(* CODESYS project Dynamixel_V3.2.2.library
   Author: Clément Jaquiéry
   Placeholder: Dynamixel
   Title: Dynamixel
   Version: 3.2.2
   Description: Permet le contrôle de Dynamixels
   Company: CPNV

Project tree, tasks and I/O mapping:
  libraries: Tc2_SerialCom, * (Beckhoff Automation GmbH); Tc2_Standard, * (Beckhoff Automation GmbH); Tc2_System, * (Beckhoff Automation GmbH); Tc2_Utilities, * (Beckhoff Automation GmbH); Tc3_Module, * (Beckhoff Automation GmbH)
  DUTs/
    data type DXL_Error
    data type E_DXL
    data type E_Packet_Status
    data type ST_DXL_Position
    data type ST_SendPacket
  GVLs/
    global variables DXL_Const
  POUs/
    function block FB_CSVRead [ST]
    function block FB_CSVWrite [ST]
    function block FB_DXL [ST]: SetActTorque, SetError, CreatePosition, DeletePosition, DisableTorque, GetActPosition, GetDatabase, Homing, MoveAbs, MovePosition, MoveRel, ReadCSV, RenamePosition, Reset, SetPosition, SetPositionD_Gain, SetPositionI_Gain, SetPositionP_Gain, SetVelocityI_Gain, SetVelocityP_Gain, ToggleTorque, WriteCSV
    function block FB_SyncDXL [ST]: AddDynamixel, ClearDynamixel, MoveAbs, MoveDiffAbs, Reset
    function block FB_U2D2_V3 [ST]: BulkWrite, BulkWriteAdd, HiByte, HiWord, LoByte, LoWord, MakeDWord, MakeWord, SendPacket, SendPacketParam, SendSyncPacket, UpdateCRC, SyncRead, SyncReadAdd, SyncWrite, SyncWriteAdd, Execute, Read, Reboot, RegWrite, SyncReset, Write
*)

// DUTs/DXL_Error
{attribute 'qualified_only'}
{attribute 'strict'}
{attribute 'to_string'}
TYPE DXL_Error :
(
	NoError := 0,
	ExceedCounter,
	ExceedTorque,
	WriteError,
	CSV_Read_Error,
	CSV_Write_Error

)BYTE;
END_TYPE

// DUTs/E_DXL
{attribute 'qualified_only'}
{attribute 'strict'}

// https://emanual.robotis.com/docs/en/dxl/x/

TYPE E_DXL :
(
	Model_Number 			:= 0, //Length 2
	Model_Information		:= 2, //Lenght 4
	Firmware_Version 		:= 6, //Length 4
	ID 						:= 7, //Length 1
	Baud_Rate 				:= 8, //Length 1
	Return_Delay_Time 		:= 9, //Length 1
	Drive_Mode 				:= 10, //Length 1
	Operating_Mode 			:= 11, //Length 1
	Secondary_ID 			:= 12, //Length 1
	Protocol_Type 			:= 13, //Length 1
	Homing_Offset 			:= 20, //Length 4
	Moving_Treshold 		:= 24, //Length 4
	Temperature_Limit 		:= 31, //Length 1
	Max_Voltage_Limit		:= 32, //Length 2
	Min_Voltage_Limit		:= 34, //Length 2
	PWM_Limit				:= 36, //Length 2
	Velocity_Limit			:= 44, //Length 4
	Max_Position_Limit		:= 48, //Length 4
	Min_Position_Limit		:= 52, //Length 4
	Startup_Configuration	:= 60, //Length 1
	Shutdown				:= 63, //Length 1
	Torque_Enable 			:= 64, //Length 1
	LED 					:= 65, //Length 1
	Status_Return_Level 	:= 68, //Length 1
	Registered_Instruction 	:= 69, //Length 1
	Hardware_Error_Status 	:= 70, //Length 1
	Velocity_I_Gain			:= 76, //Length 2
	Velocity_P_Gain			:= 78, //Length 2
	Position_D_Gain			:= 80, //Length 2
	Position_I_Gain			:= 82, //Length 2
	Position_P_Gain			:= 84, //Length 2
	Feedforward_2nd_Gain	:= 88, //Length 2
	Feedforward_1st_Gain	:= 90, //Length 2
	Bus_Watchdog			:= 98, //Length 1
	Goal_PWM				:= 100, //Length 2
	Goal_Velocity			:= 104, //Length 4
	Profile_Acceleration	:= 108, //Length 4
	Profile_Velocity		:= 112, //Length 4
	Goal_Position			:= 116, //Length 4
	Realtime_Tick			:= 120, //Length 2
	Moving					:= 122, //Length 1
	Moving_Status			:= 123, //Length 1
	Present_PWM				:= 124, //Length 2
	Present_Load			:= 126, //Length 2
	Present_Velocity		:= 128, //Length 4
	Present_Position		:= 132, //Length 4
	Velocity_Trajectory		:= 136, //Length 4
	Position_Trajectory		:= 140, //Length 4
	Present_Input_Voltage	:= 144, //Length 2
	Present_Temperature		:= 146, //Length 1
	Backup_Ready			:= 147  //Length 1
)BYTE;
END_TYPE

// DUTs/E_Packet_Status
{attribute 'qualified_only'}
{attribute 'strict'}
TYPE E_Packet_Status : 						// https://emanual.robotis.com/docs/en/dxl/protocol2/
(
	Waiting						:= 0,	
	Send_Result_Fail			:= 1,	// Failed to process the sent Instruction Packet
	Send_Instruction_Error		:= 2,	// An undefined Instruction has been used. Action has been used without Reg Write
	Send_CRC_Error				:= 3,   // The CRC of the sent Packet does not match the expected value
	Send_Data_Range_Error		:= 4,	// Data to be written to the specified Address is outside the range of the minimum/maximum value
	Send_Data_Lenght_Error		:= 5,	// Attempted to write Data that is shorter than the required data length of the specified Address (ex: when you attempt to only use 2 bytes of a register that has been defined as 4 bytes)
	Send_Data_Limit_Error		:= 6,	// Data to be written to the specified Address is outside of the configured Limit value
	Send_Access_Error			:= 7,	// Attempted to write a value to an Address that is Read Only or has not been defined. Attempted to read a value from an Address that is Write Only or has not been defined. Attempted to write a value to an EEPROM register while Torque was Enabled.
	Receive_TimeOut,
	Receive_Instruction_Error,
	Receive_CRC_Error,
	SendByte_Fail,
	Success
)BYTE;
END_TYPE

// DUTs/ST_DXL_Position
TYPE ST_DXL_Position :
STRUCT
	byIndex : BYTE;
	sName	: T_MaxString;
	diPos	: DINT;
END_STRUCT
END_TYPE

// DUTs/ST_SendPacket
TYPE ST_SendPacket :
STRUCT
	eStatus : ARRAY[0..252] OF E_Packet_Status;
	diValue : ARRAY[0..252] OF DINT;
	arPacket : ARRAY[0..MAX_PACKET_LENGTH] OF BYTE;
	wLength : WORD;
	byNumPacketsReceive : BYTE;
END_STRUCT
END_TYPE

// GVLs/DXL_Const
VAR_GLOBAL CONSTANT
	//--------------Paramètres de réglage des dynamixels--------------
	MAX_ERROR : BYTE := 5;						// Nombre d'essais de communication avant de se mettre en erreur
	TIME_TORQUE_ERROR : TIME := T#250MS;		// Temps avant que le dynamixel soit en erreur dû aux couples
	TIME_OUT_PACKET : TIME := T#100MS;			// Temps avant que le dynamixel soit en erreur dû aux non retour de paquet
	//--------------Paramètres de longueurs max de paquets--------------
	MAX_LENGTH_BUFFER : WORD := 74;				// Longueur max de la mémoire tampon d'envois de paquets
	MAX_PACKET_LENGTH : BYTE := 99;				// Longueur max des paquets envoyés
	MAX_RECEIVE_PACKET_LENGTH : WORD := 300;	// Longueur max des paquets reçus
	//--------------Paramètres de longueurs max du tableau--------------
	MAX_CSV_ROWS 			: UDINT := 29;	// |, Longueur du tableau à ajuster pour avoir plus de position
	MAX_CSV_COLUMNS 		: UDINT := 2;	// -, Ne pas toucher
	MAX_CSV_FIELD_LENGTH	: UDINT := 20;	// Ne pas toucher
END_VAR

// POUs/FB_CSVRead
FUNCTION_BLOCK FB_CSVRead(* Reading of CSV file in binary mode. Field values may contain non-printing control characters (binary data or special characters like line feed, carriage return or quotation mark...). *)
VAR	
	nRow	 	: UDINT 	:= 0;(* Row number (record) *)
	nColumn		: UDINT 	:= 0;(* Column number (record field) *)
	cbDone		: UDINT 	:= 0;(* Counts allready parsed data bytes *)
	hFile		: UINT		:= 0;(* File handle of the source file *)
	step		: DWORD 	:= 0;
	fbFileOpen	: FB_FileOpen;(* Opens file *)
	fbFileClose	: FB_FileClose;(* Closes file *)
	fbFileRead	: FB_FileRead;(* Writes binary data *)
	fbReader	: FB_CSVMemBufferReader;(* Helper function block used to parse CSV data bytes *)

	record		: ARRAY[0..1024] OF BYTE;(* Binary row data buffer. The size of this buffer have to be > length of longest record line + 2 (CRLF)  *)
	cbRecord	: UDINT := 0;(* Number of bytes in row buffer *)
	cbField		: UDINT;(* Number of bytes in field buffer *)
END_VAR
VAR_INPUT
	bRead		: BOOL := FALSE;(* Rising edge starts program execution *)
	sNetId		: T_AmsNetId := '';	(* TwinCAT system network address *)
	sFileName	: T_MaxString := '';(* CSV source file path and name *)
	database	: POINTER TO ARRAY[0..MAX_CSV_ROWS] OF ST_DXL_Position;(* Target PLC database *)
END_VAR
VAR_OUTPUT
	bBusy		: BOOL;
	bError		: BOOL;
	nErrId		: UDINT;
END_VAR

CASE step OF
	0:	(* Wait for rising edge at bRead variable *)
		IF bRead THEN
			bRead 	:= FALSE;
			bBusy 	:= TRUE;
			bError	:= FALSE;
			nErrId	:= 0;
			hFile	:= 0;
			nRow	:= 0;
			nColumn	:= 0;
			cbRecord:= 0;
			cbDone 	:= 0;
			step 	:= 1;
		END_IF

	1:	(* Open source file *)
		fbFileOpen(  bExecute := FALSE  );
		fbFileOpen( sNetId := sNetId, sPathName := sFileName, nMode := FOPEN_MODEREAD OR FOPEN_MODEBINARY,(* Open file in BINARY mode! *)
					ePath := PATH_GENERIC, bExecute := TRUE );
		step := 2;

	2:(* Wait until open not busy *)
		fbFileOpen( bExecute := FALSE, bError => bError, nErrID => nErrID, hFile => hFile );
		IF NOT fbFileOpen.bBusy THEN
			IF NOT fbFileOpen.bError THEN
				step := 3;
			ELSE(* Error: file not found? *)
				step := 100;
			END_IF
		END_IF

	3:	(* Read data bytes from file *)
		fbFileRead( bExecute := FALSE );
		fbFileRead( sNetId := sNetId, hFile := hFile, pReadBuff := ADR( record[ cbRecord ] ), cbReadLen := SIZEOF( record ) - cbRecord, bExecute :=TRUE );
		step := 4;

	4:(* Wait until read not busy *)
		fbFileRead( bExecute := FALSE, bError => bError, nErrID => nErrID );
		IF NOT fbFileRead.bBusy THEN
			IF NOT fbFileRead.bError THEN
				IF fbFileRead.bEOF THEN
					step := 10;(* End of file reached => Close source file *)
				ELSE
					cbRecord := cbRecord + fbFileRead.cbRead;(* Recalculate the new size of data buffer *)
					step := 5;(* Parse binary data *)
				END_IF
			ELSE(* Error *)
				step := 100;
			END_IF
		END_IF

	5:(* Parse binary data *)
		cbDone := 0;(* Reset number of parsed data bytes *)
		fbReader.eCmd := eEnumCmd_First;(* Read first field value *)
		REPEAT
			fbReader( pBuffer := ADR( record ), cbBuffer := cbRecord );
			IF fbReader.bOk THEN
				fbReader.eCmd := eEnumCmd_Next;(* Read next field value *)
				cbDone := cbDone + fbReader.cbRead;(* Count the number of successfully parsed data bytes *)

				IF ( nRow <= MAX_CSV_ROWS ) THEN
					(* Convert every CSV data field to PLC data field format *)
					CASE nColumn OF
						0:(* sName : T_MaxString *)
							cbField := CSVFIELD_TO_ARG( fbReader.pValue, fbReader.cbValue,  TRUE, F_BYTE( database^[nRow].byIndex ) );
						1:(* nNumber : UDINT *)
							cbField := CSVFIELD_TO_ARG( fbReader.pValue, fbReader.cbValue,  TRUE, F_STRING( database^[nRow].sName ) );
						2:(* fPos : LREAL *)
							cbField := CSVFIELD_TO_ARG( fbReader.pValue, fbReader.cbValue,  TRUE, F_DINT( database^[nRow].diPos ) );
					ELSE
						;
					END_CASE
				END_IF

				nColumn := nColumn + 1;(* Increment number of read columns *)
				IF fbReader.bCRLF THEN(* CRLF == TRUE => End of reacord reached *)
					nRow 		:= nRow + 1;(* Increment number of read records *)
					nColumn 	:= 0;(* Reset number of columns *)
				END_IF

			ELSE(* Error: End of buffer reached or all fields parsed *)
				cbRecord := MEMMOVE( ADR( record ), ADR( record[ cbDone ] ), cbRecord - cbDone );(* Shift left the remaining (not allready read) data bytes *)
				step := 3;(* Read new data bytes *)
			END_IF
		UNTIL NOT fbReader.bOk
		END_REPEAT

	10:	(* Close source file *)
		fbFileClose( bExecute := FALSE );
		fbFileClose( sNetId := sNetId, hFile := hFile, bExecute := TRUE );
		step := 11;

	11:(* Wait until close not busy *)
		fbFileClose( bExecute := FALSE, bError => bError, nErrID => nErrID );
		IF ( NOT fbFileClose.bBusy ) THEN
			hFile := 0;
			step := 100;
		END_IF

	100: (* Error or ready step => cleanup *)
		IF ( hFile <> 0 ) THEN
			step := 10; (* Close the source file *)
		ELSE
			bBusy := FALSE;
			step := 0;	(* Ready *)
		END_IF

END_CASE

END_FUNCTION_BLOCK

// POUs/FB_CSVWrite
FUNCTION_BLOCK FB_CSVWrite(* Writing of CSV file in binary mode. Field values may contain non-printing control characters (binary data or special characters like line feed, carriage return or quotation mark...). *)
VAR
	nRow	 	: UDINT 	:= 0;(* Row number (record) *)
	nColumn		: UDINT 	:= 0;(* Column number (record field) *)
	hFile		: UINT		:= 0;(* File handle of the source file *)
	step		: DWORD 	:= 0;

	fbFileOpen	: FB_FileOpen;(* Opens file *)
	fbFileClose	: FB_FileClose;(* Closes file *)
	fbFileWrite	: FB_FileWrite;(* Reads binary data *)
	fbWriter	: FB_CSVMemBufferWriter;(* Helper function block used to create CSV data bytes *)

	record		: ARRAY[0..1024] OF BYTE;(* Binary (row) data buffer. The size of this buffer have to be > length of longest record line + 2 (CRLF)  *)
	cbRecord	: UDINT := 0;(* Number of bytes in row buffer *)
	field		: ARRAY[0..MAX_CSV_FIELD_LENGTH] OF BYTE;(* Binary (field) data buffer. The size of this buffer have to be > length of the longest field *)
	cbField		: UDINT;(* Number of bytes in field buffer *)
END_VAR
VAR_INPUT
	bWrite		: BOOL := FALSE;(* Rising edge starts program execution *)
	sNetId		: T_AmsNetId := '';	(* TwinCAT system network address *)
	sFileName	: T_MaxString := '';(* CSV destination file path and name *)
	database	: POINTER TO ARRAY[0..MAX_CSV_COLUMNS ] OF ST_DXL_Position;(* Target PLC database *)
END_VAR
VAR_OUTPUT
	bBusy		: BOOL;
	bError		: BOOL;
	nErrId		: UDINT;
END_VAR

CASE step OF
	0:	(* Wait for rising edge at bWrite variable *)
		IF bWrite THEN
			bWrite 	:= FALSE;
			bBusy 	:= TRUE;
			bError	:= FALSE;
			nErrId	:= 0;
			hFile	:= 0;
			nRow	:= 0;
			nColumn := 0;
			step 	:= 1;
		END_IF

	1:	(* Open source file *)
		fbFileOpen( bExecute := FALSE  );
		fbFileOpen( sNetId := sNetId, sPathName := sFileName, nMode := FOPEN_MODEWRITE OR FOPEN_MODEBINARY, (* Open file in BINARY mode! *)
					ePath := PATH_GENERIC, bExecute := TRUE );
		step := 2;

	2:(* Wait until open not busy *)
		fbFileOpen( bExecute := FALSE, bError => bError, nErrID => nErrID, hFile => hFile );
		IF NOT fbFileOpen.bBusy THEN
			IF NOT fbFileOpen.bError THEN
				step := 3;
			ELSE(* Error: file not found? *)
				step := 100;
			END_IF
		END_IF

	3:(* Convert one PLC record to CSV format *)
		cbRecord := 0;
		fbWriter.eCmd := eEnumCmd_First;(* Write first field value *)
		IF nRow <= MAX_CSV_ROWS THEN

			(* Convert every PLC data field to the CSV data field format *)
			FOR nColumn := 0 TO MAX_CSV_COLUMNS BY 1 DO

				cbField := 0;(* Reset *)
				CASE nColumn OF
					0:(* sName : T_MaxString *)
						cbField := ARG_TO_CSVFIELD( F_BYTE( database^[ nRow ].byIndex ), TRUE, ADR( field ), SIZEOF( field ) );
					1:(* nNumber : UDINT *)
						cbField := ARG_TO_CSVFIELD( F_STRING( database^[ nRow ].sName ), TRUE, ADR( field ), SIZEOF( field ) );
					2:(* fPos : LREAL *)
						cbField := ARG_TO_CSVFIELD( F_DINT( database^[ nRow ].diPos ), TRUE, ADR( field ), SIZEOF( field ) );
				ELSE
					;
				END_CASE

				IF cbField > 0 THEN
					(* Add new field to the record buffer *)
					fbWriter( 	pBuffer := ADR( record ), cbBuffer := SIZEOF( record ), putValue :='',  pValue := ADR( field ), cbValue := cbField,
								bCRLF := ( nColumn = MAX_CSV_COLUMNS ) );(* bCRLF == TRUE => Write CRLF after the last field value *)
					IF fbWriter.bOk THEN
						fbWriter.eCmd 	:= eEnumCmd_Next;(* Write next field value *)
						cbRecord 		:= cbRecord + fbWriter.cbWrite;(* Calculate the new record size *)
					ELSE(* Error *)
						step := 100;
						RETURN;
					END_IF
				END_IF

			END_FOR(* FOR nColumn := 0... *)

			nRow := nRow + 1;(* Increment number of created records (rows) *)
			step := 4;(* Write record to the file *)

		ELSE(* All rows written => Close file *)
			step := 10;
		END_IF


	4:	(* Write record to file *)
		fbFileWrite( bExecute := FALSE );
		fbFileWrite( sNetId := sNetId, hFile := hFile, pWriteBuff := ADR( record ), cbWriteLen := cbRecord, bExecute := TRUE );
		step := 5;

	5:(* Wait until write not busy *)
		fbFileWrite( bExecute := FALSE, bError => bError, nErrID => nErrID );
		IF NOT fbFileWrite.bBusy THEN
			IF NOT fbFileWrite.bError THEN
				step := 3;(* Write next record *)
			ELSE(* Error *)
				step := 100;
			END_IF
		END_IF

	10:	(* Close source file *)
		fbFileClose( bExecute := FALSE );
		fbFileClose( sNetId := sNetId, hFile := hFile, bExecute := TRUE );
		step := 11;

	11:(* Wait until close not busy *)
		fbFileClose( bExecute := FALSE, bError => bError, nErrID => nErrID );
		IF ( NOT fbFileClose.bBusy ) THEN
			hFile := 0;
			step := 100;
		END_IF

	100: (* Error or ready step => cleanup *)
		IF ( hFile <> 0 ) THEN
			step := 10; (* Close the source file *)
		ELSE
			bBusy := FALSE;
			step := 0;	(* Ready *)
		END_IF

END_CASE

END_FUNCTION_BLOCK

// POUs/FB_DXL
FUNCTION_BLOCK FB_DXL
VAR_INPUT
	sFonction			: STRING;					// Texte pour indiquer la fonction du dynamixel ex: Bras robot droit
	ID					: BYTE(0..252);
	MaxTorque			: WORD(0..LOAD_LIMIT);		// 500 => 50% du torque maximum
	Reverse				: BOOL;						// Inversion du sens de rotation
	TorqueStartup		: BOOL;						// Torque activé au démarrage

	bHomingMode			: BOOL; // Faux = Homing par couple, vrai = homing par capteur
	bHomingSensor		: BOOL; // Si HomingMode = vrai, relier cette variable au capteur
	iHomingVelocity		: INT(-VELOCITY_LIMIT..VELOCITY_LIMIT) := 100;
	wHomingTorque		: WORD(0..LOAD_LIMIT) := 100;
	wMoveVelocity		: WORD(0..PWM_LIMIT) := 855;
	wPosTolerance		: WORD := 100;
	wPositionP_Gain		: WORD; // Gain P, de positionnement
	wPositionI_Gain		: WORD; // Gain I, de positionnement
	wPositionD_Gain		: WORD; // Gain D, de positionnement
	wVelocityP_Gain		: WORD; // Gain P, de vitesse
	wVelocityI_Gain		: WORD; // Gain I, de vitesse
END_VAR
VAR_INPUT CONSTANT
	sCSVFilePath : T_MaxString := '';
END_VAR
VAR_OUTPUT
	Init : BOOL;
	HomingDone : BOOL;
	bDatabaseNotSave : BOOL;
	diActTorque : DINT;
	Error	: BOOL;
	ErrorID : DXL_Error;
END_VAR
VAR_IN_OUT
	U2D2 : FB_U2D2_V3;
END_VAR
VAR
	stSendPacket : ST_SendPacket;
	Counter : BYTE;
	Step : BYTE;
	StepError : BYTE;
	bReset : BOOL;
	aDatabase : ARRAY[0..MAX_CSV_ROWS] OF ST_DXL_Position;
END_VAR
VAR CONSTANT
	VELOCITY_LIMIT : INT := 1023;
	LOAD_LIMIT : WORD := 1000;
	PWM_LIMIT : WORD := 855;
	EXTENDED_POSITION_LIMIT : DINT := 1048575;
END_VAR

IF Error THEN
	Counter := 0;
	Step := 0;
	CASE StepError OF
		0:
			IF U2D2.Write(ADR(stSendPacket), ID, E_DXL.Torque_Enable, 1, 0) THEN
				StepError := 1;
			END_IF

		1:
			IF stSendPacket.eStatus[0] <> E_Packet_Status.Waiting THEN
				IF stSendPacket.eStatus[0] = E_Packet_Status.Success THEN
					StepError := 2;
				ELSE
					StepError := 0;
				END_IF
			END_IF
	END_CASE
END_IF

IF NOT Init AND NOT Error THEN
	CASE Step OF
		0:
			IF U2D2.Reboot(ADR(stSendPacket), ID) THEN
				Counter := Counter + 1;
				Step := 1;
			END_IF
		1:
			IF stSendPacket.eStatus[0] <> E_Packet_Status.Waiting THEN
				IF stSendPacket.eStatus[0] = E_Packet_Status.Success THEN
					Counter := 0;
					Step := 2;
				ELSE
					Error := NOT (Counter < MAX_ERROR);
					ErrorID := DXL_Error.ExceedCounter;
					Step := 0;
				END_IF
			END_IF

		2:
			IF U2D2.Write(ADR(stSendPacket), ID, E_DXL.Torque_Enable, 1, 0)  THEN
				Counter := Counter + 1;
				Step := 3;
			END_IF
		3:
			IF stSendPacket.eStatus[0] <> E_Packet_Status.Waiting THEN
				IF stSendPacket.eStatus[0] = E_Packet_Status.Success THEN
					Counter := 0;
					Step := 4;
				ELSE
					Error := NOT (Counter < MAX_ERROR);
					ErrorID := DXL_Error.ExceedCounter;
					Step := 2;
				END_IF
			END_IF
			
		4:
			IF U2D2.Write(ADR(stSendPacket), ID, E_DXL.Drive_Mode, 1, SEL(Reverse, 2#00001000, 2#00001001)) THEN
				Counter := Counter + 1;
				Step := 5;
			END_IF
			
		5:
			IF stSendPacket.eStatus[0] <> E_Packet_Status.Waiting THEN
				IF stSendPacket.eStatus[0] = E_Packet_Status.Success THEN
					Counter := 0;
					Step := 6;
				ELSE
					Error := NOT (Counter < MAX_ERROR);
					ErrorID := DXL_Error.ExceedCounter;
					Step := 4;
				END_IF
			END_IF

		6:
			IF U2D2.Write(ADR(stSendPacket), ID, E_DXL.Startup_Configuration, 1, SEL(TorqueStartup, 2#00000000, 2#00000001)) THEN
				Counter := Counter + 1;
				Step := 7;
			END_IF

		7:
			IF stSendPacket.eStatus[0] <> E_Packet_Status.Waiting THEN
				IF stSendPacket.eStatus[0] = E_Packet_Status.Success THEN
					Counter := 0;
					Step := 8;
				ELSE
					Error := NOT (Counter < MAX_ERROR);
					ErrorID := DXL_Error.ExceedCounter;
					Step := 6;
				END_IF
			END_IF

		8:
			IF U2D2.Write(ADR(stSendPacket), ID, E_DXL.Return_Delay_Time, 1, 10) THEN
				Counter := Counter + 1;
				Step := 9;
			END_IF

		9:
			IF stSendPacket.eStatus[0] <> E_Packet_Status.Waiting THEN
				IF stSendPacket.eStatus[0] = E_Packet_Status.Success THEN
					Counter := 0;
					Step := 10;
				ELSE
					Error := NOT (Counter < MAX_ERROR);
					ErrorID := DXL_Error.ExceedCounter;
					Step := 8;
				END_IF
			END_IF

		10:
			IF TorqueStartup THEN
				IF U2D2.Write(ADR(stSendPacket), ID, E_DXL.Torque_Enable, 1, 1) THEN
					Counter := Counter + 1;
					Step := 11;
				END_IF
			ELSE
				Step := 12;
			END_IF

		11:
			IF stSendPacket.eStatus[0] <> E_Packet_Status.Waiting THEN
				IF stSendPacket.eStatus[0] = E_Packet_Status.Success THEN
					Counter := 0;
					Step := 12;
				ELSE
					Error := NOT (Counter < MAX_ERROR);
					ErrorID := DXL_Error.ExceedCounter;
					Step := 10;
				END_IF
			END_IF
			
		12: // Set PID positionnement
			IF wPositionP_Gain > 0 THEN
				IF U2D2.Write(ADR(stSendPacket), ID, E_DXL.Position_P_Gain, 2, wPositionP_Gain) THEN
					Counter := Counter + 1;
					Step := 13;
				END_IF
			ELSE
				Step := 14;
			END_IF
		
		13:
			IF stSendPacket.eStatus[0] <> E_Packet_Status.Waiting THEN
				IF stSendPacket.eStatus[0] = E_Packet_Status.Success THEN
					Counter := 0;
					Step := 14;
				ELSE
					Error := NOT (Counter < MAX_ERROR);
					ErrorID := DXL_Error.ExceedCounter;
					Step := 12;
				END_IF
			END_IF
			
		14:
			IF wPositionI_Gain > 0 THEN
				IF U2D2.Write(ADR(stSendPacket), ID, E_DXL.Position_I_Gain, 2, wPositionI_Gain) THEN
					Counter := Counter + 1;
					Step := 15;
				END_IF
			ELSE
				Step := 16;
			END_IF
		
		15:
			IF stSendPacket.eStatus[0] <> E_Packet_Status.Waiting THEN
				IF stSendPacket.eStatus[0] = E_Packet_Status.Success THEN
					Counter := 0;
					Step := 16;
				ELSE
					Error := NOT (Counter < MAX_ERROR);
					ErrorID := DXL_Error.ExceedCounter;
					Step := 14;
				END_IF
			END_IF
			
		16:
			IF wPositionD_Gain > 0 THEN
				IF U2D2.Write(ADR(stSendPacket), ID, E_DXL.Position_D_Gain, 2, wPositionD_Gain) THEN
					Counter := Counter + 1;
					Step := 17;
				END_IF
			ELSE
				Step := 18;
			END_IF
		
		17:
			IF stSendPacket.eStatus[0] <> E_Packet_Status.Waiting THEN
				IF stSendPacket.eStatus[0] = E_Packet_Status.Success THEN
					Counter := 0;
					Step := 18;
				ELSE
					Error := NOT (Counter < MAX_ERROR);
					ErrorID := DXL_Error.ExceedCounter;
					Step := 16;
				END_IF
			END_IF
			
		18: // Set gain de vitesse
			IF wVelocityP_Gain > 0 THEN
				IF U2D2.Write(ADR(stSendPacket), ID, E_DXL.Velocity_P_Gain, 2, wVelocityP_Gain) THEN
					Counter := Counter + 1;
					Step := 19;
				END_IF
			ELSE
				Step := 20;
			END_IF
		
		19:
			IF stSendPacket.eStatus[0] <> E_Packet_Status.Waiting THEN
				IF stSendPacket.eStatus[0] = E_Packet_Status.Success THEN
					Counter := 0;
					Step := 20;
				ELSE
					Error := NOT (Counter < MAX_ERROR);
					ErrorID := DXL_Error.ExceedCounter;
					Step := 18;
				END_IF
			END_IF
			
		20:
			IF wVelocityI_Gain > 0 THEN
				IF U2D2.Write(ADR(stSendPacket), ID, E_DXL.Velocity_I_Gain, 2, wVelocityI_Gain) THEN
					Counter := Counter + 1;
					Step := 21;
				END_IF
			ELSE
				Step := 22;
			END_IF
		
		21:
			IF stSendPacket.eStatus[0] <> E_Packet_Status.Waiting THEN
				IF stSendPacket.eStatus[0] = E_Packet_Status.Success THEN
					Counter := 0;
					Step := 22;
				ELSE
					Error := NOT (Counter < MAX_ERROR);
					ErrorID := DXL_Error.ExceedCounter;
					Step := 20;
				END_IF
			END_IF

		22: // Lire le tableau CSV
			IF ReadCSV() THEN
				Step := 0;
				Init := TRUE;
			END_IF
	END_CASE
END_IF

METHOD INTERNAL SetActTorque
VAR_INPUT
	_diActTorque : DINT;
END_VAR
diActTorque := _diActTorque;
END_METHOD

METHOD INTERNAL SetError
VAR_INPUT
	_Error	: BOOL;
	_ErrorID : DXL_Error;
END_VAR
Error := _Error;
ErrorID := _ErrorID;
END_METHOD

METHOD PUBLIC CreatePosition
VAR_INPUT
	byTableIndexSel : BYTE;
	diDxlPos		: DINT;
END_VAR
VAR
	udiI : UDINT;
	udiJ : UDINT;
END_VAR
IF Error OR bReset OR NOT Init THEN
	RETURN;
END_IF

// Trouver l'index qui est égal à 0
FOR udiI := 0 TO MAX_CSV_ROWS DO
	IF aDatabase[udiI].byIndex = 0 THEN
		EXIT;
	END_IF
END_FOR


IF aDatabase[udiI].byIndex = 0 THEN
	// Décaler tout les autres index qui sont égale ou plus grands que l'index séléctionné
	FOR udiJ := 0 TO MAX_CSV_ROWS DO
		IF aDatabase[udiJ].byIndex >= byTableIndexSel+1 THEN
			aDatabase[udiJ].byIndex := aDatabase[udiJ].byIndex + 1;
		END_IF
	END_FOR

	aDatabase[udiI].byIndex := byTableIndexSel+1;
	aDatabase[udiI].sName := 'Nouvelle position';
	aDatabase[udiI].diPos := diDxlPos;
	bDatabaseNotSave := TRUE;
END_IF
END_METHOD

METHOD PUBLIC DeletePosition
VAR_INPUT
	byIndex : BYTE;
END_VAR
VAR
	udiI : UDINT;
END_VAR
IF Error OR bReset OR NOT Init THEN
	RETURN;
END_IF

IF aDatabase[byIndex].byIndex <> 0 THEN
	// Décaler tout les autres index qui sont plus grands que l'index séléctionné
	FOR udiI := 0 TO MAX_CSV_ROWS DO
		IF aDatabase[udiI].byIndex > aDatabase[byIndex].byIndex THEN
			aDatabase[udiI].byIndex := aDatabase[udiI].byIndex - 1;
		END_IF
	END_FOR

	aDatabase[byIndex].byIndex := 0;
	aDatabase[byIndex].sName := '';
	aDatabase[byIndex].diPos := 0;

	bDatabaseNotSave := TRUE;
END_IF
END_METHOD

METHOD PUBLIC DisableTorque : BOOL
VAR_INST
	byStep : BYTE;
	byCounter : BYTE;
	diRead : DINT;
END_VAR
IF Error OR bReset OR NOT Init THEN
	byCounter := 0;
	byStep := 0;
	RETURN;
END_IF

{warning disable C0371}

// Vérification de la référence VAR_IN_OUT, maintien de la méthode actuelle en cas de référence invalide
IF NOT __ISVALIDREF(U2D2) THEN
     RETURN;
END_IF

CASE byStep OF
	0: // Désactiver le torque
		IF U2D2.Write(ADR(stSendPacket), ID, E_DXL.Torque_Enable, 1, 0) THEN
			byCounter := byCounter + 1;
			byStep := 1;
		END_IF

	1:
		IF stSendPacket.eStatus[0] <> E_Packet_Status.Waiting THEN
			IF stSendPacket.eStatus[0] = E_Packet_Status.Success THEN
				byCounter := 0;
				byStep := 0;
				DisableTorque := TRUE;
			ELSE
				Error := NOT (byCounter < MAX_ERROR);
				ErrorID := DXL_Error.ExceedCounter;
				byStep := 0;
			END_IF
		END_IF
END_CASE
END_METHOD

METHOD PUBLIC GetActPosition : BOOL
VAR_INST
	byStep : BYTE;
	byCounter : BYTE;
END_VAR
VAR_OUTPUT
	diPos : DINT;
END_VAR
IF Error OR bReset OR NOT Init THEN
	byCounter := 0;
	byStep := 0;
	RETURN;
END_IF

{warning disable C0371}

// Vérification de la référence VAR_IN_OUT, maintien de la méthode actuelle en cas de référence invalide
IF NOT __ISVALIDREF(U2D2) THEN
     RETURN;
END_IF

CASE byStep OF
	0:
		IF U2D2.Read(ADR(stSendPacket), ID, E_DXL.Present_Position, 4) THEN
			byCounter := byCounter + 1;
			byStep := 1;
		END_IF

	1:
		IF stSendPacket.eStatus[0] <> E_Packet_Status.Waiting THEN
			IF stSendPacket.eStatus[0] = E_Packet_Status.Success THEN
				byCounter := 0;
				diPos := stSendPacket.diValue[0];
				byStep := 0;
				GetActPosition := TRUE;
			ELSE
				Error := NOT (byCounter < MAX_ERROR);
				ErrorID := DXL_Error.ExceedCounter;
				byStep := 0;
			END_IF
		END_IF
END_CASE
END_METHOD

METHOD PUBLIC GetDatabase : ST_DXL_Position
VAR_INPUT
	byPosIndex : UDINT(0..MAX_CSV_ROWS);
END_VAR
IF bReset OR NOT Init THEN
	RETURN;
END_IF

GetDatabase := aDatabase[byPosIndex];
END_METHOD

METHOD PUBLIC Homing : BOOL
VAR
	diActTorque : DINT;
END_VAR
VAR_INST
	byStep : BYTE;
	diActPos : DINT;
	fbTimer : TON := (PT:= TIME_TORQUE_ERROR);
	diHomeOffset : DINT;
	byCounter : BYTE;
END_VAR
IF Error OR bReset OR NOT Init THEN
	byCounter := 0;
	fbTimer.IN := FALSE;
	byStep := 0;
	RETURN;
END_IF

{warning disable C0371}

// Vérification de la référence VAR_IN_OUT, maintien de la méthode actuelle en cas de référence invalide
IF NOT __ISVALIDREF(U2D2) THEN
     RETURN;
END_IF

fbTimer();

CASE byStep OF
	0:
		IF U2D2.Write(ADR(stSendPacket), ID, E_DXL.Torque_Enable, 1, 0) THEN
			byCounter := byCounter + 1;
			byStep := 1;
		END_IF

	1:
		IF stSendPacket.eStatus[0] <> E_Packet_Status.Waiting THEN
			IF stSendPacket.eStatus[0] = E_Packet_Status.Success THEN
				byCounter := 0;
				byStep := 2;
			ELSE
				Error := NOT (byCounter < MAX_ERROR);
				ErrorID := DXL_Error.ExceedCounter;
				byStep := 0;
			END_IF
		END_IF

	2:
		IF U2D2.Write(ADR(stSendPacket), ID, E_DXL.Homing_Offset, 4, 0) THEN
			byCounter := byCounter + 1;
			byStep := 3;
		END_IF

	3:
		IF stSendPacket.eStatus[0] <> E_Packet_Status.Waiting THEN
			IF stSendPacket.eStatus[0] = E_Packet_Status.Success THEN
				byCounter := 0;
				byStep := 4;
			ELSE
				Error := NOT (byCounter < MAX_ERROR);
				ErrorID := DXL_Error.ExceedCounter;
				byStep := 2;
			END_IF
		END_IF

	4:
		IF U2D2.Write(ADR(stSendPacket), ID, E_DXL.Operating_Mode, 1, 1) THEN
			byCounter := byCounter + 1;
			byStep := 5;
		END_IF

	5:
		IF stSendPacket.eStatus[0] <> E_Packet_Status.Waiting THEN
			IF stSendPacket.eStatus[0] = E_Packet_Status.Success THEN
				byCounter := 0;
				byStep := 8; //6
			ELSE
				Error := NOT (byCounter < MAX_ERROR);
				ErrorID := DXL_Error.ExceedCounter;
				byStep := 4;
			END_IF
		END_IF

	6: // Sauté grâce au bit 3 du Drive Mode
		IF U2D2.Write(ADR(stSendPacket), ID, E_DXL.Torque_Enable, 1, 1) THEN
			byCounter := byCounter + 1;
			byStep := 7;
		END_IF

	7:
		IF stSendPacket.eStatus[0] <> E_Packet_Status.Waiting THEN
			IF stSendPacket.eStatus[0] = E_Packet_Status.Success THEN
				byCounter := 0;
				byStep := 8;
			ELSE
				Error := NOT (byCounter < MAX_ERROR);
				ErrorID := DXL_Error.ExceedCounter;
				byStep := 6;
			END_IF
		END_IF

	8:
		IF U2D2.Write(ADR(stSendPacket), ID, E_DXL.Goal_Velocity, 4, INT_TO_DWORD(iHomingVelocity)) THEN
			byCounter := byCounter + 1;
			byStep := 9;
		END_IF

	9:
		IF stSendPacket.eStatus[0] <> E_Packet_Status.Waiting THEN
			IF stSendPacket.eStatus[0] = E_Packet_Status.Success THEN
				byCounter := 0;
				byStep := 10;
			ELSE
				Error := NOT (byCounter < MAX_ERROR);
				ErrorID := DXL_Error.ExceedCounter;
				byStep := 8;
			END_IF
		END_IF

	10:
		// Type de homing
		IF bHomingMode THEN
			// Par capteur
			IF bHomingSensor THEN
				byStep := 12;
			END_IF
		ELSE
			// Par couple
			IF U2D2.Read(ADR(stSendPacket), ID, E_DXL.Present_Load, 2) THEN
				byCounter := byCounter + 1;
				byStep := 11;
			END_IF
		END_IF

	11:
		IF stSendPacket.eStatus[0] <> E_Packet_Status.Waiting THEN
			IF stSendPacket.eStatus[0] = E_Packet_Status.Success THEN
				byCounter := 0;
				diActTorque := stSendPacket.diValue[0];
				IF ABS(diActTorque) >= wHomingTorque THEN
					fbTimer.IN := TRUE;
					IF fbTimer.Q THEN
						fbTimer.IN := FALSE;
						byStep := 12;
					ELSE
						byStep := 10;
					END_IF
				ELSE
					fbTimer.IN := FALSE;
					byStep := 10;
				END_IF
			ELSE
				Error := NOT (byCounter < MAX_ERROR);
				ErrorID := DXL_Error.ExceedCounter;
				byStep := 10;
			END_IF
		END_IF

	12:
		IF U2D2.Write(ADR(stSendPacket), ID, E_DXL.Goal_Velocity, 4, 0) THEN
			byCounter := byCounter + 1;
			byStep := 13;
		END_IF

	13:
		IF stSendPacket.eStatus[0] <> E_Packet_Status.Waiting THEN
			IF stSendPacket.eStatus[0] = E_Packet_Status.Success THEN
				byCounter := 0;
				byStep := 14;
			ELSE
				Error := NOT (byCounter < MAX_ERROR);
				ErrorID := DXL_Error.ExceedCounter;
				byStep := 12;
			END_IF
		END_IF

	14:
		IF U2D2.Read(ADR(stSendPacket), ID, E_DXL.Present_Position, 4) THEN
			byCounter := byCounter + 1;
			byStep := 15;
		END_IF

	15:
		IF stSendPacket.eStatus[0] <> E_Packet_Status.Waiting THEN
			IF stSendPacket.eStatus[0] = E_Packet_Status.Success THEN
				byCounter := 0;
				diActPos := stSendPacket.diValue[0];
				byStep := 16;
			ELSE
				Error := NOT (byCounter < MAX_ERROR);
				ErrorID := DXL_Error.ExceedCounter;
				byStep := 14;
			END_IF
		END_IF

	16:
		IF U2D2.Write(ADR(stSendPacket), ID, E_DXL.Torque_Enable, 1, 0) THEN
			byCounter := byCounter + 1;
			byStep := 17;
		END_IF

	17:
		IF stSendPacket.eStatus[0] <> E_Packet_Status.Waiting THEN
			IF stSendPacket.eStatus[0] = E_Packet_Status.Success THEN
				byCounter := 0;
				byStep := 18;
			ELSE
				Error := NOT (byCounter < MAX_ERROR);
				ErrorID := DXL_Error.ExceedCounter;
				byStep := 16;
			END_IF
		END_IF

	18:
		IF U2D2.Write(ADR(stSendPacket), ID, E_DXL.Homing_Offset, 4, DINT_TO_DWORD(SEL(Reverse, -diActPos, diActPos))) THEN
			byCounter := byCounter + 1;
			byStep := 19;
		END_IF

	19:
		IF stSendPacket.eStatus[0] <> E_Packet_Status.Waiting THEN
			IF stSendPacket.eStatus[0] = E_Packet_Status.Success THEN
				byCounter := 0;
				byStep := 20;
			ELSE
				Error := NOT (byCounter < MAX_ERROR);
				ErrorID := DXL_Error.ExceedCounter;
				byStep := 18;
			END_IF
		END_IF

	20:
		IF U2D2.Read(ADR(stSendPacket), ID, E_DXL.Homing_Offset, 4) THEN
			byCounter := byCounter + 1;
			byStep := 21;
		END_IF

	21: // Vérification
		IF stSendPacket.eStatus[0] <> E_Packet_Status.Waiting THEN
			IF stSendPacket.eStatus[0] = E_Packet_Status.Success THEN
				byCounter := 0;
				diHomeOffset := stSendPacket.diValue[0];
				IF SEL(Reverse, diActPos, -diActPos) = -diHomeOffset THEN
					byStep := 22;
				ELSE
					Error := TRUE;
					ErrorID := DXL_Error.WriteError;
					byStep := 0;
				END_IF
			ELSE
				Error := NOT (byCounter < MAX_ERROR);
				ErrorID := DXL_Error.ExceedCounter;
				byStep := 20;
			END_IF
		END_IF

	22:
		IF U2D2.Write(ADR(stSendPacket), ID, E_DXL.Torque_Enable, 1, 1) THEN
			byCounter := byCounter + 1;
			byStep := 23;
		END_IF

	23:
		IF stSendPacket.eStatus[0] <> E_Packet_Status.Waiting THEN
			IF stSendPacket.eStatus[0] = E_Packet_Status.Success THEN
				byCounter := 0;
				byStep := 0;
				HomingDone := TRUE;
				Homing := TRUE;
			ELSE
				Error := NOT (byCounter < MAX_ERROR);
				ErrorID := DXL_Error.ExceedCounter;
				byStep := 22;
			END_IF
		END_IF
END_CASE
END_METHOD

METHOD PUBLIC MoveAbs : BOOL
VAR_INPUT
	diPosObj : DINT(-EXTENDED_POSITION_LIMIT..EXTENDED_POSITION_LIMIT);
END_VAR
VAR
	diRead : DINT;
END_VAR
VAR_INST
	byStep : BYTE;
	byCounter : BYTE;
	fbTimer : TON := (PT:= TIME_TORQUE_ERROR);
	diReadTorque : DINT;
	diPosObjSave : DINT;
END_VAR
IF Error OR bReset OR NOT Init THEN
	byCounter := 0;
	fbTimer.IN := FALSE;
	byStep := 0;
	RETURN;
END_IF

{warning disable C0371}

// Vérification de la référence VAR_IN_OUT, maintien de la méthode actuelle en cas de référence invalide
IF NOT __ISVALIDREF(U2D2) THEN
     RETURN;
END_IF

fbTimer();

CASE byStep OF
	0:
		IF U2D2.Read(ADR(stSendPacket), ID, E_DXL.Operating_Mode, 1) THEN
			diPosObjSave := diPosObj;
			byCounter := byCounter + 1;
			byStep := 1;
		END_IF

	1:
		IF stSendPacket.eStatus[0] <> E_Packet_Status.Waiting THEN
			IF stSendPacket.eStatus[0] = E_Packet_Status.Success THEN
				byCounter := 0;
				diRead := stSendPacket.diValue[0];
				byStep := SEL(diRead = 4, 4, 2);
			ELSE
				Error := NOT (byCounter < MAX_ERROR);
				ErrorID := DXL_Error.ExceedCounter;
				byStep := 0;
			END_IF
		END_IF

	2:
		IF U2D2.Read(ADR(stSendPacket), ID, E_DXL.PWM_Limit, 2) THEN
			byCounter := byCounter + 1;
			byStep := 3;
		END_IF

	3:
		IF stSendPacket.eStatus[0] <> E_Packet_Status.Waiting THEN
			IF stSendPacket.eStatus[0] = E_Packet_Status.Success THEN
				byCounter := 0;
				diRead := stSendPacket.diValue[0];
				byStep := SEL(diRead = wMoveVelocity, 4, 12); // 10 Sauté grâce au bit 3 du Drive Mode
			ELSE
				Error := NOT (byCounter < MAX_ERROR);
				ErrorID := DXL_Error.ExceedCounter;
				byStep := 2;
			END_IF
		END_IF

	4:
		IF U2D2.Write(ADR(stSendPacket), ID, E_DXL.Torque_Enable, 1, 0) THEN
			byCounter := byCounter + 1;
			byStep := 5;
		END_IF

	5:
		IF stSendPacket.eStatus[0] <> E_Packet_Status.Waiting THEN
			IF stSendPacket.eStatus[0] = E_Packet_Status.Success THEN
				byCounter := 0;
				byStep := 6;
			ELSE
				Error := NOT (byCounter < MAX_ERROR);
				ErrorID := DXL_Error.ExceedCounter;
				byStep := 4;
			END_IF
		END_IF

	6:
		IF U2D2.Write(ADR(stSendPacket), ID, E_DXL.Operating_Mode, 1, 4) THEN
			byCounter := byCounter + 1;
			byStep := 7;
		END_IF

	7:
		IF stSendPacket.eStatus[0] <> E_Packet_Status.Waiting THEN
			IF stSendPacket.eStatus[0] = E_Packet_Status.Success THEN
				byCounter := 0;
				byStep := 8;
			ELSE
				Error := NOT (byCounter < MAX_ERROR);
				ErrorID := DXL_Error.ExceedCounter;
				byStep := 6;
			END_IF
		END_IF

	8:
		IF U2D2.Write(ADR(stSendPacket), ID, E_DXL.PWM_Limit, 2, wMoveVelocity) THEN
			byCounter := byCounter + 1;
			byStep := 9;
		END_IF

	9:
		IF stSendPacket.eStatus[0] <> E_Packet_Status.Waiting THEN
			IF stSendPacket.eStatus[0] = E_Packet_Status.Success THEN
				byCounter := 0;
				byStep := 12; // 10 Sauté grâce au bit 3 du Drive Mode
			ELSE
				Error := NOT (byCounter < MAX_ERROR);
				ErrorID := DXL_Error.ExceedCounter;
				byStep := 8;
			END_IF
		END_IF

	10: // Sauté grâce au bit 3 du Drive Mode
		IF U2D2.Write(ADR(stSendPacket), ID, E_DXL.Torque_Enable, 1, 1) THEN
			byCounter := byCounter + 1;
			byStep := 11;
		END_IF

	11: // Sauté grâce au bit 3 du Drive Mode
		IF stSendPacket.eStatus[0] <> E_Packet_Status.Waiting THEN
			IF stSendPacket.eStatus[0] = E_Packet_Status.Success THEN
				byCounter := 0;
				byStep := 12;
			ELSE
				Error := NOT (byCounter < MAX_ERROR);
				ErrorID := DXL_Error.ExceedCounter;
				byStep := 10;
			END_IF
		END_IF

	12:
		IF U2D2.Write(ADR(stSendPacket), ID, E_DXL.Goal_Position, 4, DINT_TO_DWORD(diPosObjSave)) THEN
			byCounter := byCounter + 1;
			byStep := 13;
		END_IF

	13:
		IF stSendPacket.eStatus[0] <> E_Packet_Status.Waiting THEN
			IF stSendPacket.eStatus[0] = E_Packet_Status.Success THEN
				byCounter := 0;
				byStep := 14;
			ELSE
				Error := NOT (byCounter < MAX_ERROR);
				ErrorID := DXL_Error.ExceedCounter;
				byStep := 12;
			END_IF
		END_IF

	14:
		IF U2D2.Read(ADR(stSendPacket), ID, E_DXL.Present_Position, 4) THEN
			byCounter := byCounter + 1;
			byStep := 15;
		END_IF

	15:
		IF stSendPacket.eStatus[0] <> E_Packet_Status.Waiting THEN
			IF stSendPacket.eStatus[0] = E_Packet_Status.Success THEN
				byCounter := 0;
				diRead := stSendPacket.diValue[0];
				IF diRead <= diPosObjSave + wPosTolerance AND diPosObjSave - wPosTolerance <= diRead THEN
					byStep := 0;
					diActTorque := 0;
					MoveAbs := TRUE;
				ELSE
					byStep := 16;
				END_IF
			ELSE
				Error := NOT (byCounter < MAX_ERROR);
				ErrorID := DXL_Error.ExceedCounter;
				byStep := 14;
			END_IF
		END_IF

	16: // Vérification de collision, le Torque > Torque max
		IF U2D2.Read(ADR(stSendPacket), ID, E_DXL.Present_Load, 2) THEN
			byCounter := byCounter + 1;
			byStep := 17;
		END_IF

	17:
		IF stSendPacket.eStatus[0] <> E_Packet_Status.Waiting THEN
			IF stSendPacket.eStatus[0] = E_Packet_Status.Success THEN
				byCounter := 0;
				diReadTorque := stSendPacket.diValue[0];
				diActTorque := diReadTorque;
				IF ABS(diReadTorque) > MaxTorque THEN
					fbTimer.IN := TRUE;
					IF fbTimer.Q THEN
						Error := TRUE;
						ErrorID := DXL_Error.ExceedTorque;
						byStep := 0;
					ELSE
						byStep := 14;
					END_IF
				ELSE
					fbTimer.IN := FALSE;
					byStep := 14;
				END_IF
			ELSE
				Error := NOT (byCounter < MAX_ERROR);
				ErrorID := DXL_Error.ExceedCounter;
				byStep := 16;
			END_IF
		END_IF
END_CASE
END_METHOD

METHOD PUBLIC MovePosition : BOOL
VAR_INPUT
	byPosIndex : UDINT(0..MAX_CSV_ROWS);
END_VAR
VAR_INST
	byStep : BYTE;
	byPosIndexSave : UDINT;
END_VAR
IF Error OR bReset OR NOT Init THEN
	byStep := 0;
	RETURN;
END_IF

CASE byStep OF
	0:
		IF aDatabase[byPosIndex].byIndex <> 0 THEN
			byPosIndexSave := byPosIndex;
			byStep := 1;
		END_IF

	1:
		IF MoveAbs(aDatabase[byPosIndexSave].diPos) THEN
			byStep := 0;
			MovePosition := TRUE;
		END_IF
END_CASE
END_METHOD

METHOD PUBLIC MoveRel : BOOL
VAR_INPUT
	diPosObj : DINT(-EXTENDED_POSITION_LIMIT..EXTENDED_POSITION_LIMIT);
END_VAR
VAR
	diRead : DINT;
END_VAR
VAR_INST
	byStep : BYTE;
	diDepl : DINT;
	byCounter : BYTE;
	fbTimer : TON := (PT:= TIME_TORQUE_ERROR);
	diReadTorque : DINT;
	diPosObjSave : DINT;
END_VAR
VAR CONSTANT
	TOLERANCE : BYTE := 5;
END_VAR
IF Error OR bReset OR NOT Init THEN
	byCounter := 0;
	fbTimer.IN := FALSE;
	byStep := 0;
	RETURN;
END_IF

{warning disable C0371}

// Vérification de la référence VAR_IN_OUT, maintien de la méthode actuelle en cas de référence invalide
IF NOT __ISVALIDREF(U2D2) THEN
     RETURN;
END_IF

fbTimer();

CASE byStep OF
	0:
		IF U2D2.Read(ADR(stSendPacket), ID, E_DXL.Operating_Mode, 1) THEN
			diPosObjSave := diPosObj;
			byCounter := byCounter + 1;
			byStep := 1;
		END_IF

	1:
		IF stSendPacket.eStatus[0] <> E_Packet_Status.Waiting THEN
			IF stSendPacket.eStatus[0] = E_Packet_Status.Success THEN
				byCounter := 0;
				diRead := stSendPacket.diValue[0];
				byStep := SEL(diRead = 4, 4, 2);
			ELSE
				Error := NOT (byCounter < MAX_ERROR);
				ErrorID := DXL_Error.ExceedCounter;
				byStep := 0;
			END_IF
		END_IF

	2:
		IF U2D2.Read(ADR(stSendPacket), ID, E_DXL.PWM_Limit, 2) THEN
			byCounter := byCounter + 1;
			byStep := 3;
		END_IF

	3:
		IF stSendPacket.eStatus[0] <> E_Packet_Status.Waiting THEN
			IF stSendPacket.eStatus[0] = E_Packet_Status.Success THEN
				byCounter := 0;
				diRead := stSendPacket.diValue[0];
				byStep := SEL(diRead = wMoveVelocity, 4, 12); // 10 Sauté grâce au bit 3 du Drive Mode
			ELSE
				Error := NOT (byCounter < MAX_ERROR);
				ErrorID := DXL_Error.ExceedCounter;
				byStep := 2;
			END_IF
		END_IF

	4:
		IF U2D2.Write(ADR(stSendPacket), ID, E_DXL.Torque_Enable, 1, 0) THEN
			byCounter := byCounter + 1;
			byStep := 5;
		END_IF

	5:
		IF stSendPacket.eStatus[0] <> E_Packet_Status.Waiting THEN
			IF stSendPacket.eStatus[0] = E_Packet_Status.Success THEN
				byCounter := 0;
				byStep := 6;
			ELSE
				Error := NOT (byCounter < MAX_ERROR);
				ErrorID := DXL_Error.ExceedCounter;
				byStep := 4;
			END_IF
		END_IF

	6:
		IF U2D2.Write(ADR(stSendPacket), ID, E_DXL.Operating_Mode, 1, 4) THEN
			byCounter := byCounter + 1;
			byStep := 7;
		END_IF

	7:
		IF stSendPacket.eStatus[0] <> E_Packet_Status.Waiting THEN
			IF stSendPacket.eStatus[0] = E_Packet_Status.Success THEN
				byCounter := 0;
				byStep := 8;
			ELSE
				Error := NOT (byCounter < MAX_ERROR);
				ErrorID := DXL_Error.ExceedCounter;
				byStep := 6;
			END_IF
		END_IF

	8:
		IF U2D2.Write(ADR(stSendPacket), ID, E_DXL.PWM_Limit, 2, wMoveVelocity) THEN
			byCounter := byCounter + 1;
			byStep := 9;
		END_IF

	9:
		IF stSendPacket.eStatus[0] <> E_Packet_Status.Waiting THEN
			IF stSendPacket.eStatus[0] = E_Packet_Status.Success THEN
				byCounter := 0;
				byStep := 12; // 10 Sauté grâce au bit 3 du Drive Mode
			ELSE
				Error := NOT (byCounter < MAX_ERROR);
				ErrorID := DXL_Error.ExceedCounter;
				byStep := 8;
			END_IF
		END_IF

	10: // Sauté grâce au bit 3 du Drive Mode
		IF U2D2.Write(ADR(stSendPacket), ID, E_DXL.Torque_Enable, 1, 1) THEN
			byCounter := byCounter + 1;
			byStep := 11;
		END_IF

	11: // Sauté grâce au bit 3 du Drive Mode
		IF stSendPacket.eStatus[0] <> E_Packet_Status.Waiting THEN
			IF stSendPacket.eStatus[0] = E_Packet_Status.Success THEN
				byCounter := 0;
				byStep := 12;
			ELSE
				Error := NOT (byCounter < MAX_ERROR);
				ErrorID := DXL_Error.ExceedCounter;
				byStep := 10;
			END_IF
		END_IF

	12:
		IF U2D2.Read(ADR(stSendPacket), ID, E_DXL.Present_Position, 4) THEN
			byCounter := byCounter + 1;
			byStep := 13;
		END_IF

	13:
		IF stSendPacket.eStatus[0] <> E_Packet_Status.Waiting THEN
			IF stSendPacket.eStatus[0] = E_Packet_Status.Success THEN
				byCounter := 0;
				diRead := stSendPacket.diValue[0];
				diDepl := diRead + diPosObjSave;
				byStep := 14;
			ELSE
				Error := NOT (byCounter < MAX_ERROR);
				ErrorID := DXL_Error.ExceedCounter;
				byStep := 12;
			END_IF
		END_IF

	14:
		IF U2D2.Write(ADR(stSendPacket), ID, E_DXL.Goal_Position, 4, DINT_TO_DWORD(diDepl)) THEN
			byCounter := byCounter + 1;
			byStep := 15;
		END_IF

	15:
		IF stSendPacket.eStatus[0] <> E_Packet_Status.Waiting THEN
			IF stSendPacket.eStatus[0] = E_Packet_Status.Success THEN
				byCounter := 0;
				byStep := 16;
			ELSE
				Error := NOT (byCounter < MAX_ERROR);
				ErrorID := DXL_Error.ExceedCounter;
				byStep := 14;
			END_IF
		END_IF

	16:
		IF U2D2.Read(ADR(stSendPacket), ID, E_DXL.Present_Position, 4) THEN
			byCounter := byCounter + 1;
			byStep := 17;
		END_IF

	17:
		IF stSendPacket.eStatus[0] <> E_Packet_Status.Waiting THEN
			IF stSendPacket.eStatus[0] = E_Packet_Status.Success THEN
				byCounter := 0;
				diRead := stSendPacket.diValue[0];
				IF diRead <= diDepl + TOLERANCE AND diDepl - TOLERANCE <= diRead THEN
					byStep := 0;
					diActTorque := 0;
					MoveRel := TRUE;
				ELSE
					byStep := 18;
				END_IF
			ELSE
				Error := NOT (byCounter < MAX_ERROR);
				ErrorID := DXL_Error.ExceedCounter;
				byStep := 16;
			END_IF
		END_IF

	18: // Vérification de collision, le Torque > Torque max
		IF U2D2.Read(ADR(stSendPacket), ID, E_DXL.Present_Load, 2) THEN
			byCounter := byCounter + 1;
			byStep := 19;
		END_IF

	19:
		IF stSendPacket.eStatus[0] <> E_Packet_Status.Waiting THEN
			IF stSendPacket.eStatus[0] = E_Packet_Status.Success THEN
				byCounter := 0;
				diReadTorque := stSendPacket.diValue[0];
				diActTorque := diReadTorque;
				IF ABS(diReadTorque) > MaxTorque THEN
					fbTimer.IN := TRUE;
					IF fbTimer.Q THEN
						Error := TRUE;
						ErrorID := DXL_Error.ExceedTorque;
						byStep := 0;
					ELSE
						byStep := 16;
					END_IF
				ELSE
					fbTimer.IN := FALSE;
					byStep := 16;
				END_IF
			ELSE
				Error := NOT (byCounter < MAX_ERROR);
				ErrorID := DXL_Error.ExceedCounter;
				byStep := 18;
			END_IF
		END_IF
END_CASE
END_METHOD

METHOD PUBLIC ReadCSV : BOOL

VAR_INST
	byStep : BYTE;
	fbCSVRead : FB_CSVRead := (sNetId:= '');
END_VAR
IF Error OR bReset THEN
	byStep := 0;
	RETURN;
END_IF

IF sCSVFilePath = '' THEN
	ReadCSV := TRUE;
	RETURN;
END_IF

CASE byStep OF
	
	0: // Lire le tableau CSV
		fbCSVRead.sFileName := sCSVFilePath;
		fbCSVRead.database := ADR(aDatabase);
		fbCSVRead(bRead:= TRUE);
		byStep := 1;

	1:
		fbCSVRead();
		IF NOT fbCSVRead.bBusy THEN
			IF NOT fbCSVRead.bError THEN
				byStep := 0;
				bDatabaseNotSave := FALSE;
				ReadCSV := TRUE;
			ELSE
				Error := TRUE;
				ErrorID := DXL_Error.CSV_Read_Error;
			END_IF
		END_IF
END_CASE
END_METHOD

METHOD PUBLIC RenamePosition
VAR_INPUT
	byIndex : BYTE;
	sName : T_MaxString;
END_VAR
IF Error OR bReset OR NOT Init THEN
	RETURN;
END_IF

aDatabase[byIndex].sName := sName;
bDatabaseNotSave := TRUE;
END_METHOD

METHOD PUBLIC Reset
bReset := TRUE;
StepError := 0;
MoveAbs(0);
MoveRel(0);
Homing();
ToggleTorque();
GetActPosition();
ReadCSV();
WriteCSV();
MovePosition(0);
GetDatabase(0);
CreatePosition(0, 0);
RenamePosition(0, '');
SetPosition(0, 0);
DeletePosition(0);
SetPositionP_Gain(0);
SetPositionI_Gain(0);
SetPositionD_Gain(0);
bReset := FALSE;

HomingDone := FALSE;
Step := 0;
Init := FALSE;

StepError := 0;
Error := FALSE;
ErrorID := DXL_Error.NoError;
END_METHOD

METHOD PUBLIC SetPosition
VAR_INPUT
	byIndex : BYTE;
	diPos : DINT;
END_VAR
IF Error OR bReset OR NOT Init THEN
	RETURN;
END_IF

IF aDatabase[byIndex].byIndex <> 0 THEN
	aDatabase[byIndex].diPos := diPos;
	bDatabaseNotSave := TRUE;
END_IF
END_METHOD

METHOD PUBLIC SetPositionD_Gain : BOOL
VAR_INPUT
	D_Gain : WORD;
END_VAR
VAR_INST
	byStep : BYTE;
	byCounter : BYTE;
END_VAR
IF Error OR bReset OR NOT Init THEN
	byCounter := 0;
	byStep := 0;
	RETURN;
END_IF

{warning disable C0371}

// Vérification de la référence VAR_IN_OUT, maintien de la méthode actuelle en cas de référence invalide
IF NOT __ISVALIDREF(U2D2) THEN
     RETURN;
END_IF

CASE byStep OF
	0:
		IF U2D2.Write(ADR(stSendPacket), ID, E_DXL.Position_D_Gain, 2, D_Gain) THEN
			byCounter := byCounter + 1;
			byStep := 1;
		END_IF
	
	1:
		IF stSendPacket.eStatus[0] <> E_Packet_Status.Waiting THEN
			IF stSendPacket.eStatus[0] = E_Packet_Status.Success THEN
				byCounter := 0;
				byStep := 0;
				SetPositionD_Gain := TRUE;
			ELSE
				Error := NOT (byCounter < MAX_ERROR);
				ErrorID := DXL_Error.ExceedCounter;
				byStep := 0;
			END_IF
		END_IF
END_CASE
END_METHOD

METHOD PUBLIC SetPositionI_Gain : BOOL
VAR_INPUT
	I_Gain : WORD;
END_VAR
VAR_INST
	byStep : BYTE;
	byCounter : BYTE;
END_VAR
IF Error OR bReset OR NOT Init THEN
	byCounter := 0;
	byStep := 0;
	RETURN;
END_IF

{warning disable C0371}

// Vérification de la référence VAR_IN_OUT, maintien de la méthode actuelle en cas de référence invalide
IF NOT __ISVALIDREF(U2D2) THEN
     RETURN;
END_IF

CASE byStep OF
	0:
		IF U2D2.Write(ADR(stSendPacket), ID, E_DXL.Position_I_Gain, 2, I_Gain) THEN
			byCounter := byCounter + 1;
			byStep := 1;
		END_IF
	
	1:
		IF stSendPacket.eStatus[0] <> E_Packet_Status.Waiting THEN
			IF stSendPacket.eStatus[0] = E_Packet_Status.Success THEN
				byCounter := 0;
				byStep := 0;
				SetPositionI_Gain := TRUE;
			ELSE
				Error := NOT (byCounter < MAX_ERROR);
				ErrorID := DXL_Error.ExceedCounter;
				byStep := 0;
			END_IF
		END_IF
END_CASE
END_METHOD

METHOD PUBLIC SetPositionP_Gain : BOOL
VAR_INPUT
	P_Gain : WORD;
END_VAR
VAR_INST
	byStep : BYTE;
	byCounter : BYTE;
END_VAR
IF Error OR bReset OR NOT Init THEN
	byCounter := 0;
	byStep := 0;
	RETURN;
END_IF

{warning disable C0371}

// Vérification de la référence VAR_IN_OUT, maintien de la méthode actuelle en cas de référence invalide
IF NOT __ISVALIDREF(U2D2) THEN
     RETURN;
END_IF

CASE byStep OF
	0:
		IF U2D2.Write(ADR(stSendPacket), ID, E_DXL.Position_P_Gain, 2, P_Gain) THEN
			byCounter := byCounter + 1;
			byStep := 1;
		END_IF
	
	1:
		IF stSendPacket.eStatus[0] <> E_Packet_Status.Waiting THEN
			IF stSendPacket.eStatus[0] = E_Packet_Status.Success THEN
				byCounter := 0;
				byStep := 0;
				SetPositionP_Gain := TRUE;
			ELSE
				Error := NOT (byCounter < MAX_ERROR);
				ErrorID := DXL_Error.ExceedCounter;
				byStep := 0;
			END_IF
		END_IF
END_CASE
END_METHOD

METHOD PUBLIC SetVelocityI_Gain : BOOL
VAR_INPUT
	I_Gain : WORD;
END_VAR
VAR_INST
	byStep : BYTE;
	byCounter : BYTE;
END_VAR
IF Error OR bReset OR NOT Init THEN
	byCounter := 0;
	byStep := 0;
	RETURN;
END_IF

{warning disable C0371}

// Vérification de la référence VAR_IN_OUT, maintien de la méthode actuelle en cas de référence invalide
IF NOT __ISVALIDREF(U2D2) THEN
     RETURN;
END_IF

CASE byStep OF
	0:
		IF U2D2.Write(ADR(stSendPacket), ID, E_DXL.Velocity_I_Gain, 2, I_Gain) THEN
			byCounter := byCounter + 1;
			byStep := 1;
		END_IF
	
	1:
		IF stSendPacket.eStatus[0] <> E_Packet_Status.Waiting THEN
			IF stSendPacket.eStatus[0] = E_Packet_Status.Success THEN
				byCounter := 0;
				byStep := 0;
				SetVelocityI_Gain := TRUE;
			ELSE
				Error := NOT (byCounter < MAX_ERROR);
				ErrorID := DXL_Error.ExceedCounter;
				byStep := 0;
			END_IF
		END_IF
END_CASE
END_METHOD

METHOD PUBLIC SetVelocityP_Gain : BOOL
VAR_INPUT
	P_Gain : WORD;
END_VAR
VAR_INST
	byStep : BYTE;
	byCounter : BYTE;
END_VAR
IF Error OR bReset OR NOT Init THEN
	byCounter := 0;
	byStep := 0;
	RETURN;
END_IF

{warning disable C0371}

// Vérification de la référence VAR_IN_OUT, maintien de la méthode actuelle en cas de référence invalide
IF NOT __ISVALIDREF(U2D2) THEN
     RETURN;
END_IF

CASE byStep OF
	0:
		IF U2D2.Write(ADR(stSendPacket), ID, E_DXL.Velocity_P_Gain, 2, P_Gain) THEN
			byCounter := byCounter + 1;
			byStep := 1;
		END_IF
	
	1:
		IF stSendPacket.eStatus[0] <> E_Packet_Status.Waiting THEN
			IF stSendPacket.eStatus[0] = E_Packet_Status.Success THEN
				byCounter := 0;
				byStep := 0;
				SetVelocityP_Gain := TRUE;
			ELSE
				Error := NOT (byCounter < MAX_ERROR);
				ErrorID := DXL_Error.ExceedCounter;
				byStep := 0;
			END_IF
		END_IF
END_CASE
END_METHOD

METHOD PUBLIC ToggleTorque : BOOL
VAR_INST
	byStep : BYTE;
	byCounter : BYTE;
	diRead : DINT;
END_VAR
IF Error OR bReset OR NOT Init THEN
	byCounter := 0;
	byStep := 0;
	RETURN;
END_IF

{warning disable C0371}

// Vérification de la référence VAR_IN_OUT, maintien de la méthode actuelle en cas de référence invalide
IF NOT __ISVALIDREF(U2D2) THEN
     RETURN;
END_IF

CASE byStep OF
	0:
		IF U2D2.Read(ADR(stSendPacket), ID, E_DXL.Torque_Enable, 1) THEN
			byCounter := byCounter + 1;
			byStep := 1;
		END_IF

	1:
		IF stSendPacket.eStatus[0] <> E_Packet_Status.Waiting THEN
			IF stSendPacket.eStatus[0] = E_Packet_Status.Success THEN
				byCounter := 0;
				diRead := stSendPacket.diValue[0];
				byStep := SEL(diRead = 0, 4, 2);
			ELSE
				Error := NOT (byCounter < MAX_ERROR);
				ErrorID := DXL_Error.ExceedCounter;
				byStep := 0;
			END_IF
		END_IF

	2: // Activer le torque
		IF U2D2.Write(ADR(stSendPacket), ID, E_DXL.Torque_Enable, 1, 1) THEN
			byCounter := byCounter + 1;
			byStep := 3;
		END_IF

	3:
		IF stSendPacket.eStatus[0] <> E_Packet_Status.Waiting THEN
			IF stSendPacket.eStatus[0] = E_Packet_Status.Success THEN
				byCounter := 0;
				byStep := 0;
				ToggleTorque := TRUE;
			ELSE
				Error := NOT (byCounter < MAX_ERROR);
				ErrorID := DXL_Error.ExceedCounter;
				byStep := 2;
			END_IF
		END_IF

	4: // Désactiver le torque
		IF U2D2.Write(ADR(stSendPacket), ID, E_DXL.Torque_Enable, 1, 0) THEN
			byCounter := byCounter + 1;
			byStep := 5;
		END_IF

	5:
		IF stSendPacket.eStatus[0] <> E_Packet_Status.Waiting THEN
			IF stSendPacket.eStatus[0] = E_Packet_Status.Success THEN
				byCounter := 0;
				byStep := 0;
				ToggleTorque := TRUE;
			ELSE
				Error := NOT (byCounter < MAX_ERROR);
				ErrorID := DXL_Error.ExceedCounter;
				byStep := 4;
			END_IF
		END_IF
END_CASE
END_METHOD

METHOD PUBLIC WriteCSV : BOOL

VAR_INST
	byStep : BYTE;
	fbCSVWrite : FB_CSVWrite := (sNetId:= '');
END_VAR
IF Error OR bReset OR NOT Init THEN
	byStep := 0;
	RETURN;
END_IF

IF sCSVFilePath = '' THEN
	WriteCSV := TRUE;
	RETURN;
END_IF

CASE byStep OF
	
	0: // Écrire le tableau CSV
		fbCSVWrite.sFileName := sCSVFilePath;
		fbCSVWrite.database := ADR(aDatabase);
		fbCSVWrite(bWrite:= TRUE);
		byStep := 1;

	1:
		fbCSVWrite();
		IF NOT fbCSVWrite.bBusy THEN
			IF NOT fbCSVWrite.bError THEN
				byStep := 0;
				bDatabaseNotSave := FALSE;
				WriteCSV := TRUE;
			ELSE
				Error := TRUE;
				ErrorID := DXL_Error.CSV_Write_Error;
			END_IF
		END_IF
END_CASE
END_METHOD

END_FUNCTION_BLOCK

// POUs/FB_U2D2_V3
FUNCTION_BLOCK FB_U2D2_V3
VAR_INPUT
	udiComPort : UDINT(1..255) := 1;				// Numéro port série ex: COMx [1..255]
	udiBaudrate : UDINT(9600..115200) := 115200;	// Vitesse de communication avec les Dynamixels [9600..115200]
END_VAR
VAR_OUTPUT
	bPortOpened : BOOL;					// Connection avec l'U2D2 réussie
	rBufferLoad : UDINT;				// % Utilisé du Buffer
END_VAR
VAR
	//--------------Réception de byte--------------
	fbSerialLineControlADS : SerialLineControlADS;											// FB de gestion de la communication série
	stSerialCfg : ComSerialConfig;															// Struct des paramètres de la communication série
	stTxBuffer : ComBuffer;																	// Struct des Bytes envoyé
	stRxBuffer : ComBuffer;																	// Struct des Bytes reçu
	fbReceiveByte: ReceiveByte;																// FB de gestion des paquets reçus
	abyReceiveMultiplePackets : ARRAY[0..MAX_RECEIVE_PACKET_LENGTH] OF BYTE;				// Tableau des Bytes reçus
	dwReceivedSize : DWORD;																	// Nombre de Bytes reçu
	abyLastByte : ARRAY[0..3] OF BYTE;														// 4 derniers Byte reçu
	abyReceiveParam : ARRAY[0..(MAX_RECEIVE_PACKET_LENGTH-11)] OF BYTE;						// Tableau de paramètre reçu
	byReceiveID : BYTE;																		// ID du Dynamixel reçu
	wReceiveLength : WORD;																	// Longueur du paquet reçu
	byReceiveErr : BYTE;																	// Erreur reçu
	wCheckReceiveCRC : WORD;																// CRC
	byReceivePacketNumber : BYTE;															// Nombre de paquet reçu
	wNextPacketIndex : WORD;																// Index du paquet suivant

	//--------------Création du paquet--------------
	abyBuffer : ARRAY[0..MAX_LENGTH_BUFFER] OF BYTE;										// Mémoire tampon utilisé par le bloc fonction FB_MemRingBuffer
	fbBuffer : FB_MemRingBuffer;															// Bloc de fonction pour la mémoire tampon
	abyData_write : ARRAY[0..MAX_PACKET_LENGTH] OF BYTE := [16#FF, 16#FF, 16#FD, 16#00];	// Variable contenant le paquet à envoyer
	wCRC : WORD;																			// Variable du CRC du paquet à envoyer
	abySyncParam : ARRAY[0..MAX_PACKET_LENGTH-10] OF BYTE;
	bySyncParamLength : BYTE;
	
	//--------------Envoi de byte--------------
	fbTimeOut : TON := (PT:= TIME_OUT_PACKET);												// Timer de temps max après l'envoi d'un paquet
	stPacketSended : POINTER TO ST_SendPacket;												// Struct du paquet envoyé
	fbSendData : SendData;																	// Bloc de fonction pour l'envoi de paquet
	

	//--------------Variables multiples usage--------------
	udiI : UDINT;
	udiJ : UDINT;
END_VAR
VAR CONSTANT
	//--------------Paramètres du protocole Dynamixel 3.0 (Ne pas toucher)--------------
	PKT_ID : BYTE := 4;
	PKT_LENGTH_L : BYTE := 5;
	PKT_LENGTH_H : BYTE := 6;
	PKT_INSTRUCTION : BYTE := 7;
	PKT_PARAMETER : BYTE := 8;
	PKT_ERROR : BYTE := 8;
END_VAR

// -----------------------------------------------------------------------
// Programme	: FB_Dynamixel_V3
// Auteur		: Clément Jaquiéry
// Date			: 03/04/2026
// Description	: Permet le contrôle de Dynamixel
// Amélioration : Permet de contrôler plusieurs Dynamixels en même temps
// -----------------------------------------------------------------------

fbTimeOut();

stSerialCfg.ComPort := udiComPort;
stSerialCfg.Baudrate := udiBaudrate;

fbSerialLineControlADS(
	Connect:= TRUE, 
	SerialCfg:= stSerialCfg, 
	NetId:= , 
	TimeOut:= , 
	TxBuffer:= stTxBuffer, 
	RxBuffer:= stRxBuffer, 
	PortOpened=> bPortOpened, 
	Error=> , 
	ErrorID=> , 
	Busy=> , 
	TxBufCount=> , 
	RxBufCount=> );

rBufferLoad := (fbBuffer.cbSize * 100) / MAX_LENGTH_BUFFER;

//--------------Réception de paquet--------------

REPEAT
	fbReceiveByte(RXbuffer:= stRxBuffer);

	IF fbReceiveByte.ByteReceived THEN
        abyReceiveMultiplePackets[dwReceivedSize] := fbReceiveByte.ReceivedByte;

		dwReceivedSize := dwReceivedSize + 1;
    END_IF

UNTIL NOT fbReceiveByte.ByteReceived
END_REPEAT

IF dwReceivedSize <> 0 AND stPacketSended <> 0 THEN
	FOR udiI := wNextPacketIndex TO dwReceivedSize DO
		abyLastByte[3] := abyLastByte[2];
		abyLastByte[2] := abyLastByte[1];
		abyLastByte[1] := abyLastByte[0];
		abyLastByte[0] := abyReceiveMultiplePackets[udiI];

		IF abyLastByte[3] = 16#FF AND abyLastByte[2] = 16#FF AND abyLastByte[1] = 16#FD AND abyLastByte[0] = 16#00 THEN // Header valide -> lire la suite du paquet

			byReceiveID := abyReceiveMultiplePackets[udiI + (PKT_ID - 3)];

			wReceiveLength := MakeWord(abyReceiveMultiplePackets[udiI + (PKT_LENGTH_H - 3)], abyReceiveMultiplePackets[udiI + (PKT_LENGTH_L - 3)]);

			IF abyReceiveMultiplePackets[udiI + (PKT_INSTRUCTION - 3)] <> 16#55 THEN
				// l'instruction n'est pas conforme -> Skip
				stPacketSended^.eStatus[byReceivePacketNumber] := E_Packet_Status.Receive_Instruction_Error;
				byReceivePacketNumber := byReceivePacketNumber + 1;
				CONTINUE;
			END_IF

			byReceiveErr := abyReceiveMultiplePackets[udiI + (PKT_ERROR - 3)];

			IF wReceiveLength > 4 THEN // Skip si pas de paramètre
				FOR udiJ := 0 TO wReceiveLength - 5 DO
					abyReceiveParam[udiJ] := abyReceiveMultiplePackets[udiI + (PKT_PARAMETER - 2) + udiJ];
				END_FOR

				CASE wReceiveLength-4 OF
					1:
						stPacketSended^.diValue[byReceivePacketNumber] := abyReceiveParam[0];
					2:
						stPacketSended^.diValue[byReceivePacketNumber] := WORD_TO_INT(MakeWord(abyReceiveParam[1], abyReceiveParam[0]));
					4:
						stPacketSended^.diValue[byReceivePacketNumber] := DWORD_TO_DINT(MakeDWord(MakeWord(abyReceiveParam[3], abyReceiveParam[2]), MakeWord(abyReceiveParam[1], abyReceiveParam[0])));
				END_CASE
			END_IF

			wCheckReceiveCRC := UpdateCRC(udiI-3, abyReceiveMultiplePackets, wReceiveLength+4);
			IF LoByte(wCheckReceiveCRC) <> abyReceiveMultiplePackets[udiI + PKT_PARAMETER + wReceiveLength - 6] OR HiByte(wCheckReceiveCRC) <> abyReceiveMultiplePackets[udiI + PKT_PARAMETER + wReceiveLength - 5] THEN
				// Contrôle de CRC échoué, paquet non conforme
				stPacketSended^.eStatus[byReceivePacketNumber] := E_Packet_Status.Receive_CRC_Error;
				byReceivePacketNumber := byReceivePacketNumber + 1;
				CONTINUE;
			END_IF

			// Lire les potentielles erreurs
			IF byReceiveErr <> 16#00 THEN
				CASE byReceiveErr OF
					1: // Send_Result_Fail
						stPacketSended^.eStatus[byReceivePacketNumber] := E_Packet_Status.Send_Result_Fail;
					2: // Send_Instruction_Error
						stPacketSended^.eStatus[byReceivePacketNumber] := E_Packet_Status.Send_Instruction_Error;
					3: // Send_CRC_Error
						stPacketSended^.eStatus[byReceivePacketNumber] := E_Packet_Status.Send_CRC_Error;
					4: // Send_Data_Range_Error
						stPacketSended^.eStatus[byReceivePacketNumber] := E_Packet_Status.Send_Data_Range_Error;
					5: // Send_Data_Lenght_Error
						stPacketSended^.eStatus[byReceivePacketNumber] := E_Packet_Status.Send_Data_Lenght_Error;
					6: // Send_Data_Limit_Error
						stPacketSended^.eStatus[byReceivePacketNumber] := E_Packet_Status.Send_Data_Limit_Error;
					7: // Send_Access_Error
						stPacketSended^.eStatus[byReceivePacketNumber] := E_Packet_Status.Send_Access_Error;
				END_CASE
			ELSE
				// Paquet conforme
				stPacketSended^.eStatus[byReceivePacketNumber] := E_Packet_Status.Success;
			END_IF
			
			byReceivePacketNumber := byReceivePacketNumber + 1;
			wNextPacketIndex := UDINT_TO_WORD(udiI + PKT_PARAMETER + wReceiveLength - 4);
			fbTimeOut(IN:= FALSE);
		ELSE
			CONTINUE;
		END_IF
	END_FOR
END_IF

IF stPacketSended <> 0 THEN
	IF fbTimeOut.Q THEN
		stPacketSended^.eStatus[byReceivePacketNumber] := E_Packet_Status.Receive_TimeOut;
		fbTimeOut(IN:= FALSE);
		stPacketSended := 0;
	
	ELSIF byReceivePacketNumber = stPacketSended^.byNumPacketsReceive THEN
		fbTimeOut(IN := FALSE);
		stPacketSended := 0;
		
	ELSE
		fbTimeOut(IN:= TRUE);
	END_IF
END_IF

IF stPacketSended = 0 THEN
	fbBuffer.A_RemoveHead(	pRead:= ADR(stPacketSended),
							cbRead:= SIZEOF(ADR(stPacketSended)),
							pBuffer:= ADR(abyBuffer),
							cbBuffer:= SIZEOF(abyBuffer),
							bOk=> );
	IF fbBuffer.bOk THEN
		fbSendData(
			pSendData:= ADR(stPacketSended^.arPacket), 
			Length:= stPacketSended^.wLength, 
			Busy=> , 
			Error=> , 
			TXbuffer:= stTxBuffer);
			
		IF fbSendData.Error = ComError_t.COMERROR_NOERROR THEN
			byReceivePacketNumber := 0;
			dwReceivedSize := 0;
			wNextPacketIndex := 0;
			fbTimeOut(IN:= TRUE);
			
			IF stPacketSended^.byNumPacketsReceive = 0 THEN
				// Paquet envoyé
				stPacketSended^.eStatus[byReceivePacketNumber] := E_Packet_Status.Success;
				fbTimeOut(IN := FALSE);
				stPacketSended := 0;
			END_IF
		ELSE
			stPacketSended^.eStatus[0] := E_Packet_Status.SendByte_Fail;
			stPacketSended := 0;
		END_IF
	END_IF
END_IF

METHOD PUBLIC BulkWrite : BOOL
VAR
	stSendPacket : POINTER TO ST_SendPacket;
	Param : ARRAY[0..MAX_PACKET_LENGTH-10] OF BYTE;
END_VAR
IF bySyncParamLength < 9 THEN
	RETURN;
END_IF

FOR udiI := 0 TO bySyncParamLength/9-1 DO
	Param[udiJ] := abySyncParam[udiI*9];
	Param[udiJ+1] := abySyncParam[udiI*9+1];
	Param[udiJ+2] := abySyncParam[udiI*9+2];
	Param[udiJ+3] := abySyncParam[udiI*9+3];
	Param[udiJ+4] := abySyncParam[udiI*9+4];	
	CASE MakeWord(abySyncParam[udiI*9+4], abySyncParam[udiI*9+3]) OF
		1:
			Param[udiJ+5] := abySyncParam[udiI*9+5];
			udiJ := udiJ + 6;
		2:
			Param[udiJ+5] := abySyncParam[udiI*9+5];
			Param[udiJ+6] := abySyncParam[udiI*9+6];
			udiJ := udiJ + 7;
		4:
			Param[udiJ+5] := abySyncParam[udiI*9+5];
			Param[udiJ+6] := abySyncParam[udiI*9+6];
			Param[udiJ+7] := abySyncParam[udiI*9+7];
			Param[udiJ+8] := abySyncParam[udiI*9+8];
			udiJ := udiJ + 9;
		ELSE
			RETURN;
	END_CASE
END_FOR

stSendPacket^.byNumPacketsReceive := 0;

BulkWrite := SendSyncPacket(stSendPacket, 16#93, Param, UDINT_TO_BYTE(udiJ));
END_METHOD

METHOD PUBLIC BulkWriteAdd : BOOL
VAR_INPUT
	ID : BYTE;
	Address : INT;
	Length : BYTE(1..4);
	Param : DWORD;
END_VAR
abySyncParam[bySyncParamLength] := ID;
abySyncParam[bySyncParamLength+1] := LoByte(INT_TO_WORD(Address));
abySyncParam[bySyncParamLength+2] := HiByte(INT_TO_WORD(Address));
abySyncParam[bySyncParamLength+3] := LoByte(Length);
abySyncParam[bySyncParamLength+4] := HiByte(Length);
abySyncParam[bySyncParamLength+5] := LoByte(LoWord(Param));
abySyncParam[bySyncParamLength+6] := HiByte(LoWord(Param));
abySyncParam[bySyncParamLength+7] := LoByte(HiWord(Param));
abySyncParam[bySyncParamLength+8] := HiByte(HiWord(Param));
bySyncParamLength := bySyncParamLength + 9;
END_METHOD

METHOD PRIVATE HiByte : BYTE
VAR_INPUT
	w : WORD;
END_VAR
HiByte := WORD_TO_BYTE(SHR(w, 8));
END_METHOD

METHOD PRIVATE HiWord : WORD
VAR_INPUT
	l : DWORD;
END_VAR
HiWord := DWORD_TO_WORD(SHR(l, 16));
END_METHOD

METHOD PRIVATE LoByte : BYTE
VAR_INPUT
	w : WORD;
END_VAR
LoByte := WORD_TO_BYTE(w AND 16#FF);
END_METHOD

METHOD PRIVATE LoWord : WORD
VAR_INPUT
	l : DWORD;
END_VAR
LoWord := DWORD_TO_WORD(l);
END_METHOD

METHOD PRIVATE MakeDWord : DWORD
VAR_INPUT
	a : WORD;
	b : WORD;
END_VAR
MakeDWord := a;
MakeDWord := SHL(MakeDWord, 16) + b;
END_METHOD

METHOD PRIVATE MakeWord : WORD
VAR_INPUT
	a : BYTE; //HIGH
	b : BYTE; //LOW
END_VAR
MakeWord := a;
MakeWord := SHL(MakeWord, 8) + b;
END_METHOD

METHOD PRIVATE SendPacket : BOOL
VAR_INPUT
	stSendPacket : POINTER TO ST_SendPacket;
	ID : BYTE;
	Instruction : BYTE;
END_VAR
VAR
	pSendPacket : POINTER TO POINTER TO ST_SendPacket;
END_VAR
abyData_write[PKT_ID] := ID;
abyData_write[PKT_LENGTH_L] := 3;
abyData_write[PKT_INSTRUCTION] := Instruction;

wCRC := UpdateCRC(0, abyData_write, 7);
abyData_write[8] := LoByte(wCRC);
abyData_write[9] := HiByte(wCRC);

stSendPacket^.arPacket := abyData_write;
stSendPacket^.eStatus[0] := E_Packet_Status.Waiting;
stSendPacket^.wLength := 10;
stSendPacket^.byNumPacketsReceive := SEL(ID <> 254, 0, 1);

pSendPacket := ADR(stSendPacket);

IF pSendPacket <> 0 THEN
	fbBuffer.A_AddTail( pWrite:= pSendPacket,
					cbWrite:= SIZEOF(stSendPacket),
					pBuffer:= ADR(abyBuffer),
					cbBuffer:= SIZEOF(abyBuffer),
					bOk=> SendPacket);
END_IF
END_METHOD

METHOD PRIVATE SendPacketParam : BOOL;
VAR_INPUT
	stSendPacket : POINTER TO ST_SendPacket;
	ID : BYTE;
	Instruction : BYTE;
	Address : BYTE;
	Length : BYTE;
	Param : DWORD;
END_VAR
VAR
	pSendPacket : POINTER TO POINTER TO ST_SendPacket;
END_VAR
abyData_write[PKT_ID] := ID;
abyData_write[PKT_LENGTH_L] := LoByte(Length + 5);
abyData_write[PKT_LENGTH_H] := HiByte(Length + 5);
abyData_write[PKT_INSTRUCTION] := Instruction;
abyData_write[PKT_PARAMETER] := LoByte(Address);
abyData_write[PKT_PARAMETER+1] := HiByte(Address);
abyData_write[PKT_PARAMETER+2] := LoByte(LoWord(Param));
abyData_write[PKT_PARAMETER+3] := HiByte(LoWord(Param));
abyData_write[PKT_PARAMETER+4] := LoByte(HiWord(Param));
abyData_write[PKT_PARAMETER+5] := HiByte(HiWord(Param));

wCRC := UpdateCRC(0, abyData_write, Length+9);
abyData_write[Length+10] := LoByte(wCRC);
abyData_write[Length+11] := HiByte(wCRC);

stSendPacket^.arPacket := abyData_write;
stSendPacket^.eStatus[0] := E_Packet_Status.Waiting;
stSendPacket^.wLength := 12 + Length;
stSendPacket^.byNumPacketsReceive := SEL(ID <> 254, 0, 1);

pSendPacket := ADR(stSendPacket);

IF pSendPacket <> 0 THEN
	fbBuffer.A_AddTail( pWrite:= pSendPacket,
					cbWrite:= SIZEOF(stSendPacket),
					pBuffer:= ADR(abyBuffer),
					cbBuffer:= SIZEOF(abyBuffer),
					bOk=> SendPacketParam);
END_IF
END_METHOD

METHOD PRIVATE SendSyncPacket : BOOL;
VAR_INPUT
	stSendPacket : POINTER TO ST_SendPacket;
	Instruction : BYTE;
	Param : ARRAY[0..MAX_Packet_length-10] OF BYTE;
	ParamLength : BYTE;
END_VAR
VAR
	i : BYTE;
	pSendPacket : POINTER TO POINTER TO ST_SendPacket;
END_VAR
abyData_write[PKT_ID] := 254;
abyData_write[PKT_LENGTH_L] := LoByte(ParamLength + 3);//7
abyData_write[PKT_LENGTH_H] := HiByte(ParamLength + 3);
abyData_write[PKT_INSTRUCTION] := Instruction;

FOR i := 0 TO ParamLength-1 DO
	abyData_write[PKT_PARAMETER+i] := Param[i];	
END_FOR

wCRC := UpdateCRC(0, abyData_write, ParamLength+7);
abyData_write[ParamLength+8] := LoByte(wCRC);
abyData_write[ParamLength+9] := HiByte(wCRC);

stSendPacket^.arPacket := abyData_write;
stSendPacket^.eStatus[0] := E_Packet_Status.Waiting;
stSendPacket^.wLength := 10 + ParamLength;

pSendPacket := ADR(stSendPacket);

IF pSendPacket <> 0 THEN
	fbBuffer.A_AddTail( pWrite:= pSendPacket,
					cbWrite:= SIZEOF(stSendPacket),
					pBuffer:= ADR(abyBuffer),
					cbBuffer:= SIZEOF(abyBuffer),
					bOk=> SendSyncPacket);
END_IF
END_METHOD

METHOD PRIVATE UpdateCRC : WORD
VAR_INPUT
	uiStartPacket : UDINT;
    abyData_blk_ptr : ARRAY[*] OF BYTE;
    uiData_blk_size : UDINT;
END_VAR
VAR
	wCRC_accum : WORD;
	uiI, uiJ : UDINT;
END_VAR
VAR CONSTANT
	CRC_TABLE : ARRAY[0..255] OF WORD := [
		16#0000, 16#8005, 16#800F, 16#000A, 16#801B, 16#001E, 16#0014, 16#8011,
		16#8033, 16#0036, 16#003C, 16#8039, 16#0028, 16#802D, 16#8027, 16#0022,
		16#8063, 16#0066, 16#006C, 16#8069, 16#0078, 16#807D, 16#8077, 16#0072,
		16#0050, 16#8055, 16#805F, 16#005A, 16#804B, 16#004E, 16#0044, 16#8041,
		16#80C3, 16#00C6, 16#00CC, 16#80C9, 16#00D8, 16#80DD, 16#80D7, 16#00D2,
		16#00F0, 16#80F5, 16#80FF, 16#00FA, 16#80EB, 16#00EE, 16#00E4, 16#80E1,
		16#00A0, 16#80A5, 16#80AF, 16#00AA, 16#80BB, 16#00BE, 16#00B4, 16#80B1,
		16#8093, 16#0096, 16#009C, 16#8099, 16#0088, 16#808D, 16#8087, 16#0082,
		16#8183, 16#0186, 16#018C, 16#8189, 16#0198, 16#819D, 16#8197, 16#0192,
		16#01B0, 16#81B5, 16#81BF, 16#01BA, 16#81AB, 16#01AE, 16#01A4, 16#81A1,
		16#01E0, 16#81E5, 16#81EF, 16#01EA, 16#81FB, 16#01FE, 16#01F4, 16#81F1,
		16#81D3, 16#01D6, 16#01DC, 16#81D9, 16#01C8, 16#81CD, 16#81C7, 16#01C2,
		16#0140, 16#8145, 16#814F, 16#014A, 16#815B, 16#015E, 16#0154, 16#8151,
		16#8173, 16#0176, 16#017C, 16#8179, 16#0168, 16#816D, 16#8167, 16#0162,
		16#8123, 16#0126, 16#012C, 16#8129, 16#0138, 16#813D, 16#8137, 16#0132,
		16#0110, 16#8115, 16#811F, 16#011A, 16#810B, 16#010E, 16#0104, 16#8101,
		16#8303, 16#0306, 16#030C, 16#8309, 16#0318, 16#831D, 16#8317, 16#0312,
		16#0330, 16#8335, 16#833F, 16#033A, 16#832B, 16#032E, 16#0324, 16#8321,
		16#0360, 16#8365, 16#836F, 16#036A, 16#837B, 16#037E, 16#0374, 16#8371,
		16#8353, 16#0356, 16#035C, 16#8359, 16#0348, 16#834D, 16#8347, 16#0342,
		16#03C0, 16#83C5, 16#83CF, 16#03CA, 16#83DB, 16#03DE, 16#03D4, 16#83D1,
		16#83F3, 16#03F6, 16#03FC, 16#83F9, 16#03E8, 16#83ED, 16#83E7, 16#03E2,
		16#83A3, 16#03A6, 16#03AC, 16#83A9, 16#03B8, 16#83BD, 16#83B7, 16#03B2,
		16#0390, 16#8395, 16#839F, 16#039A, 16#838B, 16#038E, 16#0384, 16#8381,
		16#0280, 16#8285, 16#828F, 16#028A, 16#829B, 16#029E, 16#0294, 16#8291,
		16#82B3, 16#02B6, 16#02BC, 16#82B9, 16#02A8, 16#82AD, 16#82A7, 16#02A2,
		16#82E3, 16#02E6, 16#02EC, 16#82E9, 16#02F8, 16#82FD, 16#82F7, 16#02F2,
		16#02D0, 16#82D5, 16#82DF, 16#02DA, 16#82CB, 16#02CE, 16#02C4, 16#82C1,
		16#8243, 16#0246, 16#024C, 16#8249, 16#0258, 16#825D, 16#8257, 16#0252,
		16#0270, 16#8275, 16#827F, 16#027A, 16#826B, 16#026E, 16#0264, 16#8261,
		16#0220, 16#8225, 16#822F, 16#022A, 16#823B, 16#023E, 16#0234, 16#8231,
		16#8213, 16#0216, 16#021C, 16#8219, 16#0208, 16#820D, 16#8207, 16#0202];
END_VAR
FOR uiJ := uiStartPacket TO uiData_blk_size + uiStartPacket DO
    uiI := (SHR(wCRC_accum, 8) XOR abyData_blk_ptr[uiJ]) AND 16#FF;
    wCRC_accum := (SHL(wCRC_accum, 8) XOR CRC_TABLE[uiI]) AND 16#FFFF;
END_FOR;

UpdateCRC := wCRC_accum;
END_METHOD

METHOD PUBLIC SyncRead : BOOL
VAR_INPUT
	stSendPacket : POINTER TO ST_SendPacket;
	Address : INT;
	Length : BYTE(1..4);
END_VAR
VAR
	Param : ARRAY[0..MAX_Packet_length-10] OF BYTE;
END_VAR
IF bySyncParamLength = 0 THEN
	RETURN;
END_IF

Param[0] := LoByte(INT_TO_WORD(Address));
Param[1] := HiByte(INT_TO_WORD(Address));
Param[2] := LoByte(Length);
Param[3] := HiByte(Length);

FOR udiI:=0 TO bySyncParamLength-1 DO
	Param[udiI+4] := abySyncParam[udiI];
END_FOR

stSendPacket^.byNumPacketsReceive := bySyncParamLength;

SyncRead := SendSyncPacket(stSendPacket, 16#82, Param, bySyncParamLength+4);
END_METHOD

METHOD PUBLIC SyncReadAdd
VAR_INPUT
	ID : BYTE;
END_VAR
abySyncParam[bySyncParamLength] := ID;
bySyncParamLength := bySyncParamLength + 1;
END_METHOD

METHOD PUBLIC SyncWrite : BOOL
VAR_INPUT
	stSendPacket : POINTER TO ST_SendPacket;
	Address : INT;
	Length : BYTE(1..4);
END_VAR
VAR
	Param : ARRAY[0..MAX_Packet_length-10] OF BYTE;
END_VAR
IF bySyncParamLength < 5 THEN
	RETURN;
END_IF

Param[0] := LoByte(INT_TO_WORD(Address));
Param[1] := HiByte(INT_TO_WORD(Address));
Param[2] := LoByte(Length);
Param[3] := HiByte(Length);
FOR udiI := 0 TO bySyncParamLength/5*(Length+1) BY (Length + 1) DO
	Param[udiI+4] := abySyncParam[udiI/(Length+1)*5];
	Param[udiI+5] := abySyncParam[udiI/(Length+1)*5+1];
	Param[udiI+6] := abySyncParam[udiI/(Length+1)*5+2];
	Param[udiI+7] := abySyncParam[udiI/(Length+1)*5+3];
	Param[udiI+8] := abySyncParam[udiI/(Length+1)*5+4];	
END_FOR

stSendPacket^.byNumPacketsReceive := 0;

SyncWrite := SendSyncPacket(stSendPacket, 16#83, Param, bySyncParamLength/5*(Length+1)+4);
END_METHOD

METHOD PUBLIC SyncWriteAdd
VAR_INPUT
	ID : BYTE;
	Param : DWORD;
END_VAR
abySyncParam[bySyncParamLength] := ID;
abySyncParam[bySyncParamLength+1] := LoByte(LoWord(Param));
abySyncParam[bySyncParamLength+2] := HiByte(LoWord(Param));
abySyncParam[bySyncParamLength+3] := LoByte(HiWord(Param));
abySyncParam[bySyncParamLength+4] := HiByte(HiWord(Param));
bySyncParamLength := bySyncParamLength + 5;
END_METHOD

METHOD PUBLIC Execute : BOOL
VAR_INPUT
	stSendPacket : POINTER TO ST_SendPacket;
	ID : BYTE; //254 = Tous les Dynamixels
END_VAR
Execute := SendPacket(stSendPacket, ID, 16#5);
END_METHOD

METHOD PUBLIC Read : BOOL
VAR_INPUT
	stSendPacket : POINTER TO ST_SendPacket;
	ID : BYTE;
	Address : INT;
	Length : BYTE(1..4);
END_VAR
IF ID = 254 THEN
	RETURN;
END_IF

Read := SendPacketParam(stSendPacket, ID, 16#2, INT_TO_BYTE(Address), 2, Length);
END_METHOD

METHOD PUBLIC Reboot : BOOL
VAR_INPUT
	stSendPacket : POINTER TO ST_SendPacket;
	ID : BYTE; //254 = Tous les Dynamixels
END_VAR
Reboot := SendPacket(stSendPacket, ID, 16#8);
END_METHOD

METHOD PUBLIC RegWrite : BOOL
VAR_INPUT
	stSendPacket : POINTER TO ST_SendPacket;
	ID : BYTE; //254 = Tous les Dynamixels
	Address : INT;
	Length : BYTE(1..4);
	Param : DWORD;
END_VAR
RegWrite := SendPacketParam(stSendPacket, ID, 16#4, INT_TO_BYTE(Address), Length, Param);
END_METHOD

METHOD PUBLIC SyncReset
bySyncParamLength := 0;
END_METHOD

METHOD PUBLIC Write : BOOL;
VAR_INPUT
	stSendPacket : POINTER TO ST_SendPacket;
	ID : BYTE; //254 = Tous les Dynamixels
	Address : INT;
	Length : BYTE(1..4);
	Param : DWORD;
END_VAR
Write := SendPacketParam(stSendPacket, ID, 16#3, INT_TO_BYTE(Address), Length, Param);
END_METHOD

END_FUNCTION_BLOCK

// POUs/FB_SyncDXL
FUNCTION_BLOCK FB_SyncDXL
VAR_OUTPUT
	Error : BOOL;
	ErrorID : DXL_Error;
END_VAR
VAR
	arSelectDxl : ARRAY[0..252] OF POINTER TO FB_DXL;
	byNbDxl : BYTE;
	stSendPacket : ST_SendPacket;
	Counter : BYTE;
	bReset : BOOL;
	aDatabase : ARRAY[0..MAX_CSV_ROWS] OF ST_DXL_Position;
END_VAR
VAR_IN_OUT
	U2D2 : FB_U2D2_V3;
END_VAR
VAR CONSTANT
	VELOCITY_LIMIT : INT := 1023;
	LOAD_LIMIT : WORD := 1000;
	PWM_LIMIT : WORD := 855;
	EXTENDED_POSITION_LIMIT : DINT := 1048575;
END_VAR

METHOD PUBLIC AddDynamixel
VAR_INPUT
	DXL : POINTER TO FB_DXL;
END_VAR
VAR
	byI : BYTE;
END_VAR
arSelectDxl[byNbDxl] := DXL;
byNbDxl := byNbDxl + 1;
END_METHOD

METHOD PUBLIC ClearDynamixel
VAR_INPUT
END_VAR
byNbDxl := 0;
END_METHOD

METHOD PUBLIC MoveAbs : BOOL
VAR_INPUT
	diPosObj : DINT(-EXTENDED_POSITION_LIMIT..EXTENDED_POSITION_LIMIT);
END_VAR
VAR
	byI : BYTE;
	bAllOk : BOOL;
	bError : BOOL;
	diRead : DINT;
END_VAR
VAR_INST
	byStep : BYTE;
	byCounter : BYTE;
	fbTimer : TON := (PT:= TIME_TORQUE_ERROR);
	diReadTorque : DINT;
	diPosObjSave : DINT;
END_VAR
IF Error OR bReset THEN
	byCounter := 0;
	fbTimer.IN := FALSE;
	byStep := 0;
	RETURN;
END_IF

IF byNbDxl = 0 THEN
	byCounter := 0;
	fbTimer.IN := FALSE;
	byStep := 0;
	RETURN;
END_IF

FOR byI := 0 TO byNbDxl - 1 DO
	IF arSelectDxl[byI]^.Error THEN
		Error := TRUE;
		byCounter := 0;
		fbTimer.IN := FALSE;
		byStep := 0;
		RETURN;
	END_IF
END_FOR

{warning disable C0371}

// Vérification de la référence VAR_IN_OUT, maintien de la méthode actuelle en cas de référence invalide
IF NOT __ISVALIDREF(U2D2) THEN
     RETURN;
END_IF

fbTimer();

CASE byStep OF
	0:
		U2D2.SyncReset();
		FOR byI := 0 TO byNbDxl - 1 DO
			U2D2.SyncReadAdd(arSelectDxl[byI]^.ID);
		END_FOR
		IF U2D2.SyncRead(ADR(stSendPacket), E_DXL.Operating_Mode, 1) THEN
			diPosObjSave := diPosObj;
			byCounter := byCounter + 1;
			byStep := 1;
		END_IF

	1:
		FOR byI := 0 TO byNbDxl - 1 DO
			IF stSendPacket.eStatus[byI] = E_Packet_Status.Waiting THEN
				EXIT;
			END_IF
			byStep := 2;
		END_FOR

	2:
		byStep := 3;
		FOR byI := 0 TO byNbDxl - 1 DO
			IF stSendPacket.eStatus[byI] <> E_Packet_Status.Success THEN
				Error := NOT (byCounter < MAX_ERROR);
				ErrorID := DXL_Error.ExceedCounter;
				byStep := 0;
				EXIT;
			END_IF
		END_FOR

	3:
		byCounter := 0;
		byStep := 4;
		FOR byI := 0 TO byNbDxl - 1 DO
			IF stSendPacket.diValue[byI] <> 4 THEN
				byStep := 8;
				EXIT;
			END_IF
		END_FOR

	4:
		U2D2.SyncReset();
		FOR byI := 0 TO byNbDxl - 1 DO
			U2D2.SyncReadAdd(arSelectDxl[byI]^.ID);
		END_FOR
		IF U2D2.SyncRead(ADR(stSendPacket), E_DXL.PWM_Limit, 2) THEN
			byCounter := byCounter + 1;
			byStep := 5;
		END_IF

	5:
		FOR byI := 0 TO byNbDxl - 1 DO
			IF stSendPacket.eStatus[byI] = E_Packet_Status.Waiting THEN
				EXIT;
			END_IF
			byStep := 6;
		END_FOR

	6:
		byStep := 7;
		FOR byI := 0 TO byNbDxl - 1 DO
			IF stSendPacket.eStatus[byI] <> E_Packet_Status.Success THEN
				Error := NOT (byCounter < MAX_ERROR);
				ErrorID := DXL_Error.ExceedCounter;
				byStep := 4;
				EXIT;
			END_IF
		END_FOR

	7:
		byCounter := 0;
		byStep := 16; // 14 Sauté grâce au bit 3 du Drive Mode
		FOR byI := 0 TO byNbDxl - 1 DO
			IF stSendPacket.diValue[byI] <> arSelectDxl[byI]^.wMoveVelocity THEN
				byStep := 8;
				EXIT;
			END_IF
		END_FOR

	8:
		U2D2.SyncReset();
		FOR byI := 0 TO byNbDxl - 1 DO
			U2D2.SyncWriteAdd(arSelectDxl[byI]^.ID, 0);
		END_FOR
		IF U2D2.SyncWrite(ADR(stSendPacket), E_DXL.Torque_Enable, 1) THEN
			byCounter := byCounter + 1;
			byStep := 9;
		END_IF

	9:
		IF stSendPacket.eStatus[0] <> E_Packet_Status.Waiting THEN
			IF stSendPacket.eStatus[0] = E_Packet_Status.Success THEN
				byCounter := 0;
				byStep := 10;
			ELSE
				Error := NOT (byCounter < MAX_ERROR);
				ErrorID := DXL_Error.ExceedCounter;
				byStep := 8;
			END_IF
		END_IF

	10:
		U2D2.SyncReset();
		FOR byI := 0 TO byNbDxl - 1 DO
			U2D2.SyncWriteAdd(arSelectDxl[byI]^.ID, 4);
		END_FOR
		IF U2D2.SyncWrite(ADR(stSendPacket), E_DXL.Operating_Mode, 1) THEN
			byCounter := byCounter + 1;
			byStep := 11;
		END_IF

	11:
		IF stSendPacket.eStatus[0] <> E_Packet_Status.Waiting THEN
			IF stSendPacket.eStatus[0] = E_Packet_Status.Success THEN
				byCounter := 0;
				byStep := 12;
			ELSE
				Error := NOT (byCounter < MAX_ERROR);
				ErrorID := DXL_Error.ExceedCounter;
				byStep := 10;
			END_IF
		END_IF

	12:
		U2D2.SyncReset();
		FOR byI := 0 TO byNbDxl - 1 DO
			U2D2.SyncWriteAdd(arSelectDxl[byI]^.ID, arSelectDxl[byI]^.wMoveVelocity);
		END_FOR
		IF U2D2.SyncWrite(ADR(stSendPacket), E_DXL.PWM_Limit, 2) THEN
			byCounter := byCounter + 1;
			byStep := 13;
		END_IF

	13:
		IF stSendPacket.eStatus[0] <> E_Packet_Status.Waiting THEN
			IF stSendPacket.eStatus[0] = E_Packet_Status.Success THEN
				byCounter := 0;
				byStep := 16; // 14 Sauté grâce au bit 3 du Drive Mode
			ELSE
				Error := NOT (byCounter < MAX_ERROR);
				ErrorID := DXL_Error.ExceedCounter;
				byStep := 12;
			END_IF
		END_IF

	14:
		// Sauté grâce au bit 3 du Drive Mode
		U2D2.SyncReset();
		FOR byI := 0 TO byNbDxl - 1 DO
			U2D2.SyncWriteAdd(arSelectDxl[byI]^.ID, 1);
		END_FOR
		IF U2D2.SyncWrite(ADR(stSendPacket), E_DXL.Torque_Enable, 1) THEN
			byCounter := byCounter + 1;
			byStep := 15;
		END_IF

	15: // Sauté grâce au bit 3 du Drive Mode
		IF stSendPacket.eStatus[0] <> E_Packet_Status.Waiting THEN
			IF stSendPacket.eStatus[0] = E_Packet_Status.Success THEN
				byCounter := 0;
				byStep := 16;
			ELSE
				Error := NOT (byCounter < MAX_ERROR);
				ErrorID := DXL_Error.ExceedCounter;
				byStep := 14;
			END_IF
		END_IF

	16:
		U2D2.SyncReset();
		FOR byI := 0 TO byNbDxl - 1 DO
			U2D2.SyncWriteAdd(arSelectDxl[byI]^.ID, DINT_TO_DWORD(diPosObjSave));
		END_FOR
		IF U2D2.SyncWrite(ADR(stSendPacket), E_DXL.Goal_Position, 4) THEN
			byCounter := byCounter + 1;
			byStep := 17;
		END_IF

	17:
		IF stSendPacket.eStatus[0] <> E_Packet_Status.Waiting THEN
			IF stSendPacket.eStatus[0] = E_Packet_Status.Success THEN
				byCounter := 0;
				byStep := 18;
			ELSE
				Error := NOT (byCounter < MAX_ERROR);
				ErrorID := DXL_Error.ExceedCounter;
				byStep := 16;
			END_IF
		END_IF

	18:
		U2D2.SyncReset();
		FOR byI := 0 TO byNbDxl - 1 DO
			U2D2.SyncReadAdd(arSelectDxl[byI]^.ID);
		END_FOR
		IF U2D2.SyncRead(ADR(stSendPacket), E_DXL.Present_Position, 4) THEN
			byCounter := byCounter + 1;
			byStep := 19;
		END_IF

	19:
		FOR byI := 0 TO byNbDxl - 1 DO
			IF stSendPacket.eStatus[byI] = E_Packet_Status.Waiting THEN
				EXIT;
			END_IF
			byStep := 20;
		END_FOR

	20:
		byStep := 21;
		FOR byI := 0 TO byNbDxl - 1 DO
			IF stSendPacket.eStatus[byI] <> E_Packet_Status.Success THEN
				Error := NOT (byCounter < MAX_ERROR);
				ErrorID := DXL_Error.ExceedCounter;
				byStep := 18;
				EXIT;
			END_IF
		END_FOR

	21:
		byCounter := 0;
		byStep := 0;
		MoveAbs := TRUE;
		FOR byI := 0 TO byNbDxl - 1 DO
			diRead := stSendPacket.diValue[byI];
			IF NOT (diRead <= diPosObjSave + arSelectDxl[byI]^.wPosTolerance AND diPosObjSave - arSelectDxl[byI]^.wPosTolerance <= diRead) THEN
				MoveAbs := FALSE;
				byStep := 22;
				EXIT;
			ELSE
				arSelectDxl[byI]^.SetActTorque(0);
			END_IF
		END_FOR

	22:
		// Vérification de collision, le Torque > Torque max
		U2D2.SyncReset();
		FOR byI := 0 TO byNbDxl - 1 DO
			U2D2.SyncReadAdd(arSelectDxl[byI]^.ID);
		END_FOR
		IF U2D2.SyncRead(ADR(stSendPacket), E_DXL.Present_Load, 2) THEN
			byCounter := byCounter + 1;
			byStep := 23;
		END_IF

	23:
		FOR byI := 0 TO byNbDxl - 1 DO
			IF stSendPacket.eStatus[byI] = E_Packet_Status.Waiting THEN
				EXIT;
			END_IF
			byStep := 24;
		END_FOR

	24:
		byStep := 25;
		FOR byI := 0 TO byNbDxl - 1 DO
			IF stSendPacket.eStatus[byI] <> E_Packet_Status.Success THEN
				Error := NOT (byCounter < MAX_ERROR);
				ErrorID := DXL_Error.ExceedCounter;
				byStep := 22;
				EXIT;
			END_IF
		END_FOR

	25:
		byCounter := 0;
		fbTimer.IN := FALSE;
		byStep := 18;
		FOR byI := 0 TO byNbDxl - 1 DO
			diReadTorque := stSendPacket.diValue[byI];
			arSelectDxl[byI]^.SetActTorque(diReadTorque);
			IF ABS(diReadTorque) > arSelectDxl[byI]^.MaxTorque THEN
				fbTimer.IN := TRUE;
				IF fbTimer.Q THEN
					arSelectDxl[byI]^.SetError(TRUE, DXL_Error.ExceedTorque);
					Error := TRUE;
					ErrorID := DXL_Error.ExceedTorque;
					FOR byI := 0 TO byNbDxl - 1 DO
						IF NOT arSelectDxl[byI]^.Error THEN
							arSelectDxl[byI]^.Reset();
						END_IF
					END_FOR
					byStep := 0;
				END_IF
				EXIT;
			END_IF
		END_FOR
END_CASE
END_METHOD

METHOD PUBLIC MoveDiffAbs : BOOL
VAR_INPUT
	diPosObj : ARRAY[*] OF DINT;
END_VAR
VAR
	byI : BYTE;
	bAllOk : BOOL;
	bError : BOOL;
	diRead : DINT;
END_VAR
VAR_INST
	byStep : BYTE;
	byCounter : BYTE;
	fbTimer : TON := (PT:= TIME_TORQUE_ERROR);
	diReadTorque : DINT;
	diPosObjSave : ARRAY[0..252] OF DINT(-EXTENDED_POSITION_LIMIT..EXTENDED_POSITION_LIMIT);
END_VAR
IF Error OR bReset THEN
	byCounter := 0;
	fbTimer.IN := FALSE;
	byStep := 0;
	RETURN;
END_IF

IF byNbDxl = 0 THEN
	byCounter := 0;
	fbTimer.IN := FALSE;
	byStep := 0;
	RETURN;
END_IF

FOR byI := 0 TO byNbDxl - 1 DO
	IF arSelectDxl[byI]^.Error THEN
		Error := TRUE;
		byCounter := 0;
		fbTimer.IN := FALSE;
		byStep := 0;
		RETURN;
	END_IF
END_FOR

{warning disable C0371}

// Vérification de la référence VAR_IN_OUT, maintien de la méthode actuelle en cas de référence invalide
IF NOT __ISVALIDREF(U2D2) THEN
     RETURN;
END_IF

fbTimer();

CASE byStep OF
	0:
		U2D2.SyncReset();
		FOR byI := 0 TO byNbDxl - 1 DO
			U2D2.SyncReadAdd(arSelectDxl[byI]^.ID);
		END_FOR
		IF U2D2.SyncRead(ADR(stSendPacket), E_DXL.Operating_Mode, 1) THEN
			FOR byI := TO_BYTE(LOWER_BOUND(diPosObj, 1)) TO TO_BYTE(UPPER_BOUND(diPosObj, 1)) DO
				diPosObjSave[byI] := diPosObj[byI];
			END_FOR
			byCounter := byCounter + 1;
			byStep := 1;
		END_IF

	1:
		FOR byI := 0 TO byNbDxl - 1 DO
			IF stSendPacket.eStatus[byI] = E_Packet_Status.Waiting THEN
				EXIT;
			END_IF
			byStep := 2;
		END_FOR

	2:
		byStep := 3;
		FOR byI := 0 TO byNbDxl - 1 DO
			IF stSendPacket.eStatus[byI] <> E_Packet_Status.Success THEN
				Error := NOT (byCounter < MAX_ERROR);
				ErrorID := DXL_Error.ExceedCounter;
				byStep := 0;
				EXIT;
			END_IF
		END_FOR

	3:
		byCounter := 0;
		byStep := 4;
		FOR byI := 0 TO byNbDxl - 1 DO
			IF stSendPacket.diValue[byI] <> 4 THEN
				byStep := 8;
				EXIT;
			END_IF
		END_FOR

	4:
		U2D2.SyncReset();
		FOR byI := 0 TO byNbDxl - 1 DO
			U2D2.SyncReadAdd(arSelectDxl[byI]^.ID);
		END_FOR
		IF U2D2.SyncRead(ADR(stSendPacket), E_DXL.PWM_Limit, 2) THEN
			byCounter := byCounter + 1;
			byStep := 5;
		END_IF

	5:
		FOR byI := 0 TO byNbDxl - 1 DO
			IF stSendPacket.eStatus[byI] = E_Packet_Status.Waiting THEN
				EXIT;
			END_IF
			byStep := 6;
		END_FOR

	6:
		byStep := 7;
		FOR byI := 0 TO byNbDxl - 1 DO
			IF stSendPacket.eStatus[byI] <> E_Packet_Status.Success THEN
				Error := NOT (byCounter < MAX_ERROR);
				ErrorID := DXL_Error.ExceedCounter;
				byStep := 4;
				EXIT;
			END_IF
		END_FOR

	7:
		byCounter := 0;
		byStep := 16; // 14 Sauté grâce au bit 3 du Drive Mode
		FOR byI := 0 TO byNbDxl - 1 DO
			IF stSendPacket.diValue[byI] <> arSelectDxl[byI]^.wMoveVelocity THEN
				byStep := 8;
				EXIT;
			END_IF
		END_FOR

	8:
		U2D2.SyncReset();
		FOR byI := 0 TO byNbDxl - 1 DO
			U2D2.SyncWriteAdd(arSelectDxl[byI]^.ID, 0);
		END_FOR
		IF U2D2.SyncWrite(ADR(stSendPacket), E_DXL.Torque_Enable, 1) THEN
			byCounter := byCounter + 1;
			byStep := 9;
		END_IF

	9:
		IF stSendPacket.eStatus[0] <> E_Packet_Status.Waiting THEN
			IF stSendPacket.eStatus[0] = E_Packet_Status.Success THEN
				byCounter := 0;
				byStep := 10;
			ELSE
				Error := NOT (byCounter < MAX_ERROR);
				ErrorID := DXL_Error.ExceedCounter;
				byStep := 8;
			END_IF
		END_IF

	10:
		U2D2.SyncReset();
		FOR byI := 0 TO byNbDxl - 1 DO
			U2D2.SyncWriteAdd(arSelectDxl[byI]^.ID, 4);
		END_FOR
		IF U2D2.SyncWrite(ADR(stSendPacket), E_DXL.Operating_Mode, 1) THEN
			byCounter := byCounter + 1;
			byStep := 11;
		END_IF

	11:
		IF stSendPacket.eStatus[0] <> E_Packet_Status.Waiting THEN
			IF stSendPacket.eStatus[0] = E_Packet_Status.Success THEN
				byCounter := 0;
				byStep := 12;
			ELSE
				Error := NOT (byCounter < MAX_ERROR);
				ErrorID := DXL_Error.ExceedCounter;
				byStep := 10;
			END_IF
		END_IF

	12:
		U2D2.SyncReset();
		FOR byI := 0 TO byNbDxl - 1 DO
			U2D2.SyncWriteAdd(arSelectDxl[byI]^.ID, arSelectDxl[byI]^.wMoveVelocity);
		END_FOR
		IF U2D2.SyncWrite(ADR(stSendPacket), E_DXL.PWM_Limit, 2) THEN
			byCounter := byCounter + 1;
			byStep := 13;
		END_IF

	13:
		IF stSendPacket.eStatus[0] <> E_Packet_Status.Waiting THEN
			IF stSendPacket.eStatus[0] = E_Packet_Status.Success THEN
				byCounter := 0;
				byStep := 16; // 14 Sauté grâce au bit 3 du Drive Mode
			ELSE
				Error := NOT (byCounter < MAX_ERROR);
				ErrorID := DXL_Error.ExceedCounter;
				byStep := 12;
			END_IF
		END_IF

	14:
		// Sauté grâce au bit 3 du Drive Mode
		U2D2.SyncReset();
		FOR byI := 0 TO byNbDxl - 1 DO
			U2D2.SyncWriteAdd(arSelectDxl[byI]^.ID, 1);
		END_FOR
		IF U2D2.SyncWrite(ADR(stSendPacket), E_DXL.Torque_Enable, 1) THEN
			byCounter := byCounter + 1;
			byStep := 15;
		END_IF

	15: // Sauté grâce au bit 3 du Drive Mode
		IF stSendPacket.eStatus[0] <> E_Packet_Status.Waiting THEN
			IF stSendPacket.eStatus[0] = E_Packet_Status.Success THEN
				byCounter := 0;
				byStep := 16;
			ELSE
				Error := NOT (byCounter < MAX_ERROR);
				ErrorID := DXL_Error.ExceedCounter;
				byStep := 14;
			END_IF
		END_IF

	16:
		U2D2.SyncReset();
		FOR byI := 0 TO byNbDxl - 1 DO
			U2D2.SyncWriteAdd(arSelectDxl[byI]^.ID, DINT_TO_DWORD(diPosObjSave[byI]));
		END_FOR
		IF U2D2.SyncWrite(ADR(stSendPacket), E_DXL.Goal_Position, 4) THEN
			byCounter := byCounter + 1;
			byStep := 17;
		END_IF

	17:
		IF stSendPacket.eStatus[0] <> E_Packet_Status.Waiting THEN
			IF stSendPacket.eStatus[0] = E_Packet_Status.Success THEN
				byCounter := 0;
				byStep := 18;
			ELSE
				Error := NOT (byCounter < MAX_ERROR);
				ErrorID := DXL_Error.ExceedCounter;
				byStep := 16;
			END_IF
		END_IF

	18:
		U2D2.SyncReset();
		FOR byI := 0 TO byNbDxl - 1 DO
			U2D2.SyncReadAdd(arSelectDxl[byI]^.ID);
		END_FOR
		IF U2D2.SyncRead(ADR(stSendPacket), E_DXL.Present_Position, 4) THEN
			byCounter := byCounter + 1;
			byStep := 19;
		END_IF

	19:
		FOR byI := 0 TO byNbDxl - 1 DO
			IF stSendPacket.eStatus[byI] = E_Packet_Status.Waiting THEN
				EXIT;
			END_IF
			byStep := 20;
		END_FOR

	20:
		byStep := 21;
		FOR byI := 0 TO byNbDxl - 1 DO
			IF stSendPacket.eStatus[byI] <> E_Packet_Status.Success THEN
				Error := NOT (byCounter < MAX_ERROR);
				ErrorID := DXL_Error.ExceedCounter;
				byStep := 18;
				EXIT;
			END_IF
		END_FOR

	21:
		byCounter := 0;
		byStep := 0;
		MoveDiffAbs := TRUE;
		FOR byI := 0 TO byNbDxl - 1 DO
			diRead := stSendPacket.diValue[byI];
			IF NOT (diRead <= diPosObjSave[byI] + arSelectDxl[byI]^.wPosTolerance AND diPosObjSave[byI] - arSelectDxl[byI]^.wPosTolerance <= diRead) THEN
				MoveDiffAbs := FALSE;
				byStep := 22;
				EXIT;
			ELSE
				arSelectDxl[byI]^.SetActTorque(0);
			END_IF
		END_FOR

	22:
		// Vérification de collision, le Torque > Torque max
		U2D2.SyncReset();
		FOR byI := 0 TO byNbDxl - 1 DO
			U2D2.SyncReadAdd(arSelectDxl[byI]^.ID);
		END_FOR
		IF U2D2.SyncRead(ADR(stSendPacket), E_DXL.Present_Load, 2) THEN
			byCounter := byCounter + 1;
			byStep := 23;
		END_IF

	23:
		FOR byI := 0 TO byNbDxl - 1 DO
			IF stSendPacket.eStatus[byI] = E_Packet_Status.Waiting THEN
				EXIT;
			END_IF
			byStep := 24;
		END_FOR

	24:
		byStep := 25;
		FOR byI := 0 TO byNbDxl - 1 DO
			IF stSendPacket.eStatus[byI] <> E_Packet_Status.Success THEN
				Error := NOT (byCounter < MAX_ERROR);
				ErrorID := DXL_Error.ExceedCounter;
				byStep := 22;
				EXIT;
			END_IF
		END_FOR

	25:
		byCounter := 0;
		fbTimer.IN := FALSE;
		byStep := 18;
		FOR byI := 0 TO byNbDxl - 1 DO
			diReadTorque := stSendPacket.diValue[byI];
			arSelectDxl[byI]^.SetActTorque(diReadTorque);
			IF ABS(diReadTorque) > arSelectDxl[byI]^.MaxTorque THEN
				fbTimer.IN := TRUE;
				IF fbTimer.Q THEN
					arSelectDxl[byI]^.SetError(TRUE, DXL_Error.ExceedTorque);
					Error := TRUE;
					ErrorID := DXL_Error.ExceedTorque;
					FOR byI := 0 TO byNbDxl - 1 DO
						IF NOT arSelectDxl[byI]^.Error THEN
							arSelectDxl[byI]^.Reset();
						END_IF
					END_FOR
					byStep := 0;
				END_IF
				EXIT;
			END_IF
		END_FOR
END_CASE
END_METHOD

METHOD PUBLIC Reset
VAR_INPUT
END_VAR
VAR
	byI : BYTE;
END_VAR
bReset := TRUE;
MoveAbs(0);
bReset := FALSE;

Error := FALSE;

IF byNbDxl > 0 THEN
	FOR byI := 0 TO byNbDxl - 1 DO
		arSelectDxl[byI]^.Reset();
	END_FOR
END_IF
END_METHOD

END_FUNCTION_BLOCK
